LIN {X 0,Y 573.278,Z 350.069,A -85,B 0,C 180,E1 -2306.518,E2 -2306.518} C_VEL
LIN {X 0,Y 573.237,Z 350.076,A -85,B 0,C 180,E1 -2309.114,E2 -2309.114} C_VEL
LIN {X 0,Y 573.257,Z 350.077,A -85,B 0,C 180,E1 -2311.968,E2 -2311.968} C_VEL
LIN {X 0,Y 573.248,Z 350.072,A -85,B 0,C 180,E1 -2314.59,E2 -2314.59} C_VEL
LIN {X 0,Y 573.231,Z 350.084,A -85,B 0,C 180,E1 -2317.662,E2 -2317.662} C_VEL
LIN {X 0,Y 573.249,Z 350.078,A -85,B 0,C 180,E1 -2319.923,E2 -2319.923} C_VEL
LIN {X 0,Y 573.255,Z 350.073,A -85,B 0,C 180,E1 -2322.988,E2 -2322.988} C_VEL
LIN {X 0,Y 573.263,Z 350.076,A -85,B 0,C 180,E1 -2325.807,E2 -2325.807} C_VEL
LIN {X 0,Y 573.273,Z 350.07,A -85,B 0,C 180,E1 -2328.734,E2 -2328.734} C_VEL
LIN {X 0,Y 573.299,Z 350.074,A -85,B 0,C 180,E1 -2331.541,E2 -2331.541} C_VEL
LIN {X 0,Y 573.285,Z 350.068,A -85,B 0,C 180,E1 -2334.372,E2 -2334.372} C_VEL
LIN {X 0,Y 573.301,Z 350.068,A -85,B 0,C 180,E1 -2337.893,E2 -2337.893} C_VEL
LIN {X 0,Y 573.331,Z 350.064,A -85,B 0,C 180,E1 -2340.703,E2 -2340.703} C_VEL
LIN {X 0,Y 573.238,Z 350.08,A -85,B 0,C 180,E1 -2343.515,E2 -2343.515} C_VEL
LIN {X 0,Y 573.289,Z 350.072,A -85,B 0,C 180,E1 -2345.628,E2 -2345.628} C_VEL
LIN {X 0,Y 573.3,Z 350.067,A -85,B 0,C 180,E1 -2348.459,E2 -2348.459} C_VEL
LIN {X 0,Y 573.29,Z 350.075,A -85,B 0,C 180,E1 -2351.312,E2 -2351.312} C_VEL
LIN {X 0,Y 573.272,Z 350.071,A -85,B 0,C 180,E1 -2354.425,E2 -2354.425} C_VEL
LIN {X 0,Y 573.253,Z 350.082,A -85,B 0,C 180,E1 -2357.112,E2 -2357.112} C_VEL
LIN {X 0,Y 573.251,Z 350.072,A -85,B 0,C 180,E1 -2360.077,E2 -2360.077} C_VEL
LIN {X 0,Y 573.264,Z 350.078,A -85,B 0,C 180,E1 -2363.154,E2 -2363.154} C_VEL
LIN {X 0,Y 573.248,Z 350.074,A -85,B 0,C 180,E1 -2364.404,E2 -2364.404} C_VEL
LIN {X 0,Y 572.617,Z 350.161,A -85,B 0,C 180,E1 -2364.99,E2 -2364.99} C_VEL
LIN {X 0,Y 569.778,Z 350.515,A -85,B 0,C 180,E1 -2365.942,E2 -2365.942} C_VEL
LIN {X 0,Y 567.353,Z 350.815,A -85,B 0,C 180,E1 -2366.708,E2 -2366.708} C_VEL
LIN {X 0,Y 566.302,Z 350.944,A -85,B 0,C 180,E1 -2367.299,E2 -2367.299} C_VEL
LIN {X 0,Y 566.212,Z 350.952,A -85,B 0,C 180,E1 -2367.5,E2 -2367.5} C_VEL
LIN {X 0,Y 566.184,Z 350.958,A -85,B 0,C 180,E1 -2370.593,E2 -2370.593} C_VEL
LIN {X 0,Y 566.224,Z 350.953,A -85,B 0,C 180,E1 -2373.102,E2 -2373.102} C_VEL
LIN {X 0,Y 566.208,Z 350.951,A -85,B 0,C 180,E1 -2375.689,E2 -2375.689} C_VEL
LIN {X 0,Y 566.213,Z 350.955,A -85,B 0,C 180,E1 -2378.56,E2 -2378.56} C_VEL
LIN {X 0,Y 566.209,Z 350.954,A -85,B 0,C 180,E1 -2381.137,E2 -2381.137} C_VEL
LIN {X 0,Y 566.199,Z 350.953,A -85,B 0,C 180,E1 -2384.036,E2 -2384.036} C_VEL
LIN {X 0,Y 566.203,Z 350.955,A -85,B 0,C 180,E1 -2387.083,E2 -2387.083} C_VEL
LIN {X 0,Y 566.227,Z 350.949,A -85,B 0,C 180,E1 -2389.804,E2 -2389.804} C_VEL
LIN {X 0,Y 566.199,Z 350.962,A -85,B 0,C 180,E1 -2392.6,E2 -2392.6} C_VEL
LIN {X 0,Y 566.277,Z 351.069,A -85,B 0,C 180,E1 -2395.593,E2 -2395.593} C_VEL
LIN {X 0,Y 566.349,Z 357.943,A -85,B 0,C 180,E1 -2396.907,E2 -2396.907} C_VEL
LIN {X 0,Y 566.272,Z 373.418,A -85,B 0,C 180,E1 -2399.826,E2 -2399.826} C_VEL
LIN {X 0,Y 566.238,Z 374.613,A -85,B 0,C 180,E1 -2400.049,E2 -2400.049} C_VEL
LIN {X 0,Y 567.194,Z 381.693,A -85,B 0,C 180,E1 -2400.172,E2 -2400.172} C_VEL
LIN {X 0,Y 566.953,Z 481.195,A -85,B 0,C 180,E1 -2401.453,E2 -2401.453} C_VEL
LIN {X 0,Y 566.809,Z 494.766,A -85,B 0,C 180,E1 -2401.78,E2 -2401.78} C_VEL
LIN {X 0,Y 566.75,Z 507.497,A -85,B 0,C 180,E1 -2402.239,E2 -2402.239} C_VEL
LIN {X 0,Y 566.582,Z 518.434,A -85,B 0,C 180,E1 -2402.768,E2 -2402.768} C_VEL
LIN {X 0,Y 566.484,Z 529.803,A -85,B 0,C 180,E1 -2403.473,E2 -2403.473} C_VEL
LIN {X 0,Y 566.32,Z 539.973,A -85,B 0,C 180,E1 -2404.257,E2 -2404.257} C_VEL
LIN {X 0,Y 566.196,Z 548.312,A -85,B 0,C 180,E1 -2405.038,E2 -2405.038} C_VEL
LIN {X 0,Y 566.102,Z 556.91,A -85,B 0,C 180,E1 -2406.01,E2 -2406.01} C_VEL
LIN {X 0,Y 566.043,Z 564.378,A -85,B 0,C 180,E1 -2407.053,E2 -2407.053} C_VEL
LIN {X 0,Y 565.962,Z 570.591,A -85,B 0,C 180,E1 -2408.129,E2 -2408.129} C_VEL
LIN {X 0,Y 565.903,Z 575.802,A -85,B 0,C 180,E1 -2409.272,E2 -2409.272} C_VEL
LIN {X 0,Y 565.869,Z 579.731,A -85,B 0,C 180,E1 -2410.408,E2 -2410.408} C_VEL
LIN {X 0,Y 565.855,Z 581.723,A -85,B 0,C 180,E1 -2411.161,E2 -2411.161} C_VEL
LIN {X 0,Y 565.839,Z 583.2,A -85,B 0,C 180,E1 -2411.91,E2 -2411.91} C_VEL
LIN {X 0,Y 565.858,Z 584.57,A -85,B 0,C 180,E1 -2413.01,E2 -2413.01} C_VEL
LIN {X 0,Y 565.812,Z 584.985,A -85,B 0,C 180,E1 -2414.142,E2 -2414.142} C_VEL
LIN {X 0,Y 565.807,Z 584.704,A -85,B 0,C 180,E1 -2414.88,E2 -2414.88} C_VEL
LIN {X 0,Y 565.855,Z 583.986,A -85,B 0,C 180,E1 -2415.645,E2 -2415.645} C_VEL
LIN {X 0,Y 565.867,Z 582.912,A -85,B 0,C 180,E1 -2416.351,E2 -2416.351} C_VEL
LIN {X 0,Y 565.879,Z 580.421,A -85,B 0,C 180,E1 -2417.447,E2 -2417.447} C_VEL
LIN {X 0,Y 565.917,Z 576.904,A -85,B 0,C 180,E1 -2418.539,E2 -2418.539} C_VEL
LIN {X 0,Y 565.931,Z 572.283,A -85,B 0,C 180,E1 -2419.627,E2 -2419.627} C_VEL
LIN {X 0,Y 565.993,Z 565.294,A -85,B 0,C 180,E1 -2420.891,E2 -2420.891} C_VEL
LIN {X 0,Y 566.112,Z 557.744,A -85,B 0,C 180,E1 -2421.972,E2 -2421.972} C_VEL
LIN {X 0,Y 566.169,Z 550.08,A -85,B 0,C 180,E1 -2422.87,E2 -2422.87} C_VEL
LIN {X 0,Y 566.319,Z 540.76,A -85,B 0,C 180,E1 -2423.766,E2 -2423.766} C_VEL
LIN {X 0,Y 566.44,Z 530.463,A -85,B 0,C 180,E1 -2424.572,E2 -2424.572} C_VEL
LIN {X 0,Y 566.547,Z 519.075,A -85,B 0,C 180,E1 -2425.286,E2 -2425.286} C_VEL
LIN {X 0,Y 566.732,Z 507.128,A -85,B 0,C 180,E1 -2425.867,E2 -2425.867} C_VEL
LIN {X 0,Y 566.819,Z 493.96,A -85,B 0,C 180,E1 -2426.335,E2 -2426.335} C_VEL
LIN {X 0,Y 566.934,Z 480.736,A -85,B 0,C 180,E1 -2426.647,E2 -2426.647} C_VEL
LIN {X 0,Y 567.081,Z 379.638,A -85,B 0,C 180,E1 -2427.947,E2 -2427.947} C_VEL
LIN {X 0,Y 566.248,Z 374.594,A -85,B 0,C 180,E1 -2428.044,E2 -2428.044} C_VEL
LIN {X 0,Y 566.341,Z 358.556,A -85,B 0,C 180,E1 -2431.067,E2 -2431.067} C_VEL
LIN {X 0,Y 566.465,Z 352.939,A -85,B 0,C 180,E1 -2432.133,E2 -2432.133} C_VEL
LIN {X 0,Y 566.263,Z 350.949,A -85,B 0,C 180,E1 -2432.534,E2 -2432.534} C_VEL
LIN {X 0,Y 566.262,Z 350.95,A -85,B 0,C 180,E1 -2435.698,E2 -2435.698} C_VEL
LIN {X 0,Y 566.212,Z 350.95,A -85,B 0,C 180,E1 -2438.566,E2 -2438.566} C_VEL
LIN {X 0,Y 566.249,Z 350.954,A -85,B 0,C 180,E1 -2441.454,E2 -2441.454} C_VEL
LIN {X 0,Y 566.241,Z 350.946,A -85,B 0,C 180,E1 -2444.506,E2 -2444.506} C_VEL
LIN {X 0,Y 566.205,Z 350.961,A -85,B 0,C 180,E1 -2447.331,E2 -2447.331} C_VEL
LIN {X 0,Y 566.212,Z 350.949,A -85,B 0,C 180,E1 -2450.337,E2 -2450.337} C_VEL
LIN {X 0,Y 566.194,Z 350.959,A -85,B 0,C 180,E1 -2453.403,E2 -2453.403} C_VEL
LIN {X 0,Y 566.218,Z 350.951,A -85,B 0,C 180,E1 -2455.748,E2 -2455.748} C_VEL
LIN {X 0,Y 566.205,Z 350.95,A -85,B 0,C 180,E1 -2458.201,E2 -2458.201} C_VEL
LIN {X 0,Y 566.202,Z 350.959,A -85,B 0,C 180,E1 -2461.077,E2 -2461.077} C_VEL
LIN {X 0,Y 566.214,Z 350.951,A -85,B 0,C 180,E1 -2463.733,E2 -2463.733} C_VEL
LIN {X 0,Y 566.218,Z 350.951,A -85,B 0,C 180,E1 -2466.568,E2 -2466.568} C_VEL
LIN {X 0,Y 566.213,Z 350.951,A -85,B 0,C 180,E1 -2469.685,E2 -2469.685} C_VEL
LIN {X 0,Y 566.213,Z 350.949,A -85,B 0,C 180,E1 -2472.086,E2 -2472.086} C_VEL
LIN {X 0,Y 566.172,Z 350.965,A -85,B 0,C 180,E1 -2475.035,E2 -2475.035} C_VEL
LIN {X 0,Y 566.214,Z 350.949,A -85,B 0,C 180,E1 -2477.912,E2 -2477.912} C_VEL
LIN {X 0,Y 566.219,Z 350.955,A -85,B 0,C 180,E1 -2480.726,E2 -2480.726} C_VEL
LIN {X 0,Y 566.214,Z 350.949,A -85,B 0,C 180,E1 -2483.782,E2 -2483.782} C_VEL
LIN {X 0,Y 566.207,Z 350.951,A -85,B 0,C 180,E1 -2486.265,E2 -2486.265} C_VEL
LIN {X 0,Y 566.195,Z 350.961,A -85,B 0,C 180,E1 -2488.921,E2 -2488.921} C_VEL
LIN {X 0,Y 566.222,Z 350.948,A -85,B 0,C 180,E1 -2491.858,E2 -2491.858} C_VEL
LIN {X 0,Y 566.219,Z 350.951,A -85,B 0,C 180,E1 -2494.251,E2 -2494.251} C_VEL
LIN {X 0,Y 566.186,Z 350.962,A -85,B 0,C 180,E1 -2496.712,E2 -2496.712} C_VEL
LIN {X 0,Y 566.213,Z 350.949,A -85,B 0,C 180,E1 -2499.662,E2 -2499.662} C_VEL
LIN {X 0,Y 566.198,Z 350.961,A -85,B 0,C 180,E1 -2502.668,E2 -2502.668} C_VEL
LIN {X 0,Y 566.225,Z 350.948,A -85,B 0,C 180,E1 -2505.626,E2 -2505.626} C_VEL
LIN {X 0,Y 566.266,Z 350.953,A -85,B 0,C 180,E1 -2508.654,E2 -2508.654} C_VEL
LIN {X 0,Y 566.24,Z 350.946,A -85,B 0,C 180,E1 -2511.434,E2 -2511.434} C_VEL
LIN {X 0,Y 566.253,Z 350.95,A -85,B 0,C 180,E1 -2514.301,E2 -2514.301} C_VEL
LIN {X 0,Y 566.272,Z 350.943,A -85,B 0,C 180,E1 -2517.866,E2 -2517.866} C_VEL
LIN {X 0,Y 566.299,Z 350.945,A -85,B 0,C 180,E1 -2520.711,E2 -2520.711} C_VEL
LIN {X 0,Y 566.27,Z 350.946,A -85,B 0,C 180,E1 -2522.845,E2 -2522.845} C_VEL
LIN {X 0,Y 566.252,Z 350.945,A -85,B 0,C 180,E1 -2525.698,E2 -2525.698} C_VEL
LIN {X 0,Y 566.239,Z 350.954,A -85,B 0,C 180,E1 -2528.565,E2 -2528.565} C_VEL
LIN {X 0,Y 566.241,Z 350.946,A -85,B 0,C 180,E1 -2531.454,E2 -2531.454} C_VEL
LIN {X 0,Y 566.224,Z 350.956,A -85,B 0,C 180,E1 -2534.507,E2 -2534.507} C_VEL
LIN {X 0,Y 566.196,Z 350.951,A -85,B 0,C 180,E1 -2537.332,E2 -2537.332} C_VEL
LIN {X 0,Y 566.212,Z 350.959,A -85,B 0,C 180,E1 -2540.337,E2 -2540.337} C_VEL
LIN {X 0,Y 566.182,Z 350.953,A -85,B 0,C 180,E1 -2543.404,E2 -2543.404} C_VEL
LIN {X 0,Y 566.217,Z 350.951,A -85,B 0,C 180,E1 -2545.749,E2 -2545.749} C_VEL
LIN {X 0,Y 566.2,Z 350.961,A -85,B 0,C 180,E1 -2548.204,E2 -2548.204} C_VEL
LIN {X 0,Y 566.187,Z 350.956,A -85,B 0,C 180,E1 -2550.592,E2 -2550.592} C_VEL
LIN {X 0,Y 566.222,Z 350.948,A -85,B 0,C 180,E1 -2553.102,E2 -2553.102} C_VEL
LIN {X 0,Y 566.205,Z 350.953,A -85,B 0,C 180,E1 -2555.689,E2 -2555.689} C_VEL
LIN {X 0,Y 566.211,Z 350.952,A -85,B 0,C 180,E1 -2558.56,E2 -2558.56} C_VEL
LIN {X 0,Y 566.208,Z 350.95,A -85,B 0,C 180,E1 -2561.137,E2 -2561.137} C_VEL
LIN {X 0,Y 566.196,Z 350.962,A -85,B 0,C 180,E1 -2564.036,E2 -2564.036} C_VEL
LIN {X 0,Y 566.201,Z 350.951,A -85,B 0,C 180,E1 -2567.083,E2 -2567.083} C_VEL
LIN {X 0,Y 566.225,Z 350.955,A -85,B 0,C 180,E1 -2569.804,E2 -2569.804} C_VEL
LIN {X 0,Y 566.197,Z 350.952,A -85,B 0,C 180,E1 -2572.6,E2 -2572.6} C_VEL
LIN {X 0,Y 566.221,Z 350.949,A -85,B 0,C 180,E1 -2575.184,E2 -2575.184} C_VEL
LIN {X 0,Y 566.234,Z 350.954,A -85,B 0,C 180,E1 -2577.744,E2 -2577.744} C_VEL
LIN {X 0,Y 566.228,Z 350.952,A -85,B 0,C 180,E1 -2580.324,E2 -2580.324} C_VEL
LIN {X 0,Y 566.219,Z 350.951,A -85,B 0,C 180,E1 -2582.662,E2 -2582.662} C_VEL
LIN {X 0,Y 566.237,Z 350.95,A -85,B 0,C 180,E1 -2585.04,E2 -2585.04} C_VEL
LIN {X 0,Y 566.233,Z 351.027,A -85,B 0,C 180,E1 -2585.919,E2 -2585.919} C_VEL
LIN {X 0,Y 567.201,Z 357.146,A -85,B 0,C 180,E1 -2586.834,E2 -2586.834} C_VEL
LIN {X 0,Y 566.963,Z 376.072,A -85,B 0,C 180,E1 -2589.502,E2 -2589.502} C_VEL
LIN {X 0,Y 566.667,Z 397.345,A -85,B 0,C 180,E1 -2592.497,E2 -2592.497} C_VEL
LIN {X 0,Y 566.459,Z 419.948,A -85,B 0,C 180,E1 -2595.633,E2 -2595.633} C_VEL
LIN {X 0,Y 566.417,Z 422.524,A -85,B 0,C 180,E1 -2595.987,E2 -2595.987} C_VEL
LIN {X 0,Y 567.226,Z 430.323,A -85,B 0,C 180,E1 -2596.11,E2 -2596.11} C_VEL
LIN {X 0,Y 566.964,Z 530.961,A -85,B 0,C 180,E1 -2597.403,E2 -2597.403} C_VEL
LIN {X 0,Y 566.871,Z 544.228,A -85,B 0,C 180,E1 -2597.72,E2 -2597.72} C_VEL
LIN {X 0,Y 566.74,Z 556.383,A -85,B 0,C 180,E1 -2598.148,E2 -2598.148} C_VEL
LIN {X 0,Y 566.589,Z 568.449,A -85,B 0,C 180,E1 -2598.724,E2 -2598.724} C_VEL
LIN {X 0,Y 566.442,Z 580.203,A -85,B 0,C 180,E1 -2599.455,E2 -2599.455} C_VEL
LIN {X 0,Y 566.321,Z 590.605,A -85,B 0,C 180,E1 -2600.266,E2 -2600.266} C_VEL
LIN {X 0,Y 566.207,Z 599.115,A -85,B 0,C 180,E1 -2601.074,E2 -2601.074} C_VEL
LIN {X 0,Y 566.112,Z 606.962,A -85,B 0,C 180,E1 -2601.972,E2 -2601.972} C_VEL
LIN {X 0,Y 566.003,Z 614.623,A -85,B 0,C 180,E1 -2603.047,E2 -2603.047} C_VEL
LIN {X 0,Y 566.004,Z 621.68,A -85,B 0,C 180,E1 -2604.299,E2 -2604.299} C_VEL
LIN {X 0,Y 565.933,Z 626.373,A -85,B 0,C 180,E1 -2605.37,E2 -2605.37} C_VEL
LIN {X 0,Y 565.927,Z 629.958,A -85,B 0,C 180,E1 -2606.44,E2 -2606.44} C_VEL
LIN {X 0,Y 565.878,Z 631.808,A -85,B 0,C 180,E1 -2607.153,E2 -2607.153} C_VEL
LIN {X 0,Y 565.846,Z 634.185,A -85,B 0,C 180,E1 -2608.577,E2 -2608.577} C_VEL
LIN {X 0,Y 565.839,Z 635,A -85,B 0,C 180,E1 -2610,E2 -2610} C_VEL
LIN {X 0,Y 565.846,Z 634.186,A -85,B 0,C 180,E1 -2611.423,E2 -2611.423} C_VEL
LIN {X 0,Y 565.878,Z 631.81,A -85,B 0,C 180,E1 -2612.847,E2 -2612.847} C_VEL
LIN {X 0,Y 565.926,Z 628.896,A -85,B 0,C 180,E1 -2613.916,E2 -2613.916} C_VEL
LIN {X 0,Y 565.878,Z 624.949,A -85,B 0,C 180,E1 -2614.987,E2 -2614.987} C_VEL
LIN {X 0,Y 566.002,Z 619.868,A -85,B 0,C 180,E1 -2616.058,E2 -2616.058} C_VEL
LIN {X 0,Y 566.04,Z 613.469,A -85,B 0,C 180,E1 -2617.132,E2 -2617.132} C_VEL
LIN {X 0,Y 566.133,Z 605.479,A -85,B 0,C 180,E1 -2618.207,E2 -2618.207} C_VEL
LIN {X 0,Y 566.228,Z 597.337,A -85,B 0,C 180,E1 -2619.105,E2 -2619.105} C_VEL
LIN {X 0,Y 566.343,Z 587.403,A -85,B 0,C 180,E1 -2620.005,E2 -2620.005} C_VEL
LIN {X 0,Y 566.529,Z 576.294,A -85,B 0,C 180,E1 -2620.807,E2 -2620.807} C_VEL
LIN {X 0,Y 566.612,Z 565.181,A -85,B 0,C 180,E1 -2621.446,E2 -2621.446} C_VEL
LIN {X 0,Y 566.736,Z 552.989,A -85,B 0,C 180,E1 -2621.988,E2 -2621.988} C_VEL
LIN {X 0,Y 566.91,Z 540.187,A -85,B 0,C 180,E1 -2622.393,E2 -2622.393} C_VEL
LIN {X 0,Y 566.997,Z 528.125,A -85,B 0,C 180,E1 -2622.641,E2 -2622.641} C_VEL
LIN {X 0,Y 567.065,Z 426.951,A -85,B 0,C 180,E1 -2623.937,E2 -2623.937} C_VEL
LIN {X 0,Y 566.435,Z 422.441,A -85,B 0,C 180,E1 -2624.024,E2 -2624.024} C_VEL
LIN {X 0,Y 566.648,Z 399.148,A -85,B 0,C 180,E1 -2627.251,E2 -2627.251} C_VEL
LIN {X 0,Y 566.926,Z 378.732,A -85,B 0,C 180,E1 -2630.121,E2 -2630.121} C_VEL
LIN {X 0,Y 567.199,Z 357.118,A -85,B 0,C 180,E1 -2633.166,E2 -2633.166} C_VEL
LIN {X 0,Y 566.236,Z 350.957,A -85,B 0,C 180,E1 -2634.105,E2 -2634.105} C_VEL
LIN {X 0,Y 566.209,Z 350.954,A -85,B 0,C 180,E1 -2636.659,E2 -2636.659} C_VEL
LIN {X 0,Y 566.196,Z 350.953,A -85,B 0,C 180,E1 -2638.952,E2 -2638.952} C_VEL
LIN {X 0,Y 566.203,Z 350.952,A -85,B 0,C 180,E1 -2641.42,E2 -2641.42} C_VEL
LIN {X 0,Y 566.212,Z 350.957,A -85,B 0,C 180,E1 -2643.955,E2 -2643.955} C_VEL
LIN {X 0,Y 566.215,Z 350.952,A -85,B 0,C 180,E1 -2646.568,E2 -2646.568} C_VEL
LIN {X 0,Y 566.212,Z 350.954,A -85,B 0,C 180,E1 -2649.685,E2 -2649.685} C_VEL
LIN {X 0,Y 566.211,Z 350.957,A -85,B 0,C 180,E1 -2652.086,E2 -2652.086} C_VEL
LIN {X 0,Y 566.169,Z 350.955,A -85,B 0,C 180,E1 -2655.035,E2 -2655.035} C_VEL
LIN {X 0,Y 566.214,Z 350.956,A -85,B 0,C 180,E1 -2658.135,E2 -2658.135} C_VEL
LIN {X 0,Y 566.218,Z 350.949,A -85,B 0,C 180,E1 -2660.727,E2 -2660.727} C_VEL
LIN {X 0,Y 566.211,Z 350.959,A -85,B 0,C 180,E1 -2663.783,E2 -2663.783} C_VEL
LIN {X 0,Y 566.222,Z 350.95,A -85,B 0,C 180,E1 -2666.262,E2 -2666.262} C_VEL
LIN {X 0,Y 566.196,Z 350.952,A -85,B 0,C 180,E1 -2668.921,E2 -2668.921} C_VEL
LIN {X 0,Y 566.189,Z 350.953,A -85,B 0,C 180,E1 -2671.046,E2 -2671.046} C_VEL
LIN {X 0,Y 566.237,Z 350.953,A -85,B 0,C 180,E1 -2673.46,E2 -2673.46} C_VEL
LIN {X 0,Y 566.19,Z 350.96,A -85,B 0,C 180,E1 -2675.819,E2 -2675.819} C_VEL
LIN {X 0,Y 566.208,Z 350.95,A -85,B 0,C 180,E1 -2678.902,E2 -2678.902} C_VEL
LIN {X 0,Y 566.205,Z 350.954,A -85,B 0,C 180,E1 -2681.172,E2 -2681.172} C_VEL
LIN {X 0,Y 566.213,Z 350.956,A -85,B 0,C 180,E1 -2683.412,E2 -2683.412} C_VEL
LIN {X 0,Y 566.191,Z 350.952,A -85,B 0,C 180,E1 -2686.359,E2 -2686.359} C_VEL
LIN {X 0,Y 566.265,Z 350.943,A -85,B 0,C 180,E1 -2688.654,E2 -2688.654} C_VEL
LIN {X 0,Y 566.241,Z 350.955,A -85,B 0,C 180,E1 -2691.435,E2 -2691.435} C_VEL
LIN {X 0,Y 566.253,Z 350.945,A -85,B 0,C 180,E1 -2694.302,E2 -2694.302} C_VEL
LIN {X 0,Y 566.272,Z 350.944,A -85,B 0,C 180,E1 -2697.866,E2 -2697.866} C_VEL
LIN {X 0,Y 566.3,Z 350.94,A -85,B 0,C 180,E1 -2700.711,E2 -2700.711} C_VEL
LIN {X 0,Y 566.272,Z 350.944,A -85,B 0,C 180,E1 -2702.846,E2 -2702.846} C_VEL
LIN {X 0,Y 566.256,Z 350.947,A -85,B 0,C 180,E1 -2705.699,E2 -2705.699} C_VEL
LIN {X 0,Y 566.242,Z 350.946,A -85,B 0,C 180,E1 -2708.566,E2 -2708.566} C_VEL
LIN {X 0,Y 566.242,Z 350.95,A -85,B 0,C 180,E1 -2711.455,E2 -2711.455} C_VEL
LIN {X 0,Y 566.225,Z 350.949,A -85,B 0,C 180,E1 -2714.508,E2 -2714.508} C_VEL
LIN {X 0,Y 566.197,Z 350.958,A -85,B 0,C 180,E1 -2717.332,E2 -2717.332} C_VEL
LIN {X 0,Y 566.213,Z 350.949,A -85,B 0,C 180,E1 -2720.337,E2 -2720.337} C_VEL
LIN {X 0,Y 566.223,Z 350.951,A -85,B 0,C 180,E1 -2723.403,E2 -2723.403} C_VEL
LIN {X 0,Y 566.219,Z 350.949,A -85,B 0,C 180,E1 -2725.749,E2 -2725.749} C_VEL
LIN {X 0,Y 566.212,Z 350.952,A -85,B 0,C 180,E1 -2727.5,E2 -2727.5} C_VEL
LIN {X 0,Y 565.531,Z 351.036,A -85,B 0,C 180,E1 -2728.093,E2 -2728.093} C_VEL
LIN {X 0,Y 562.66,Z 351.4,A -85,B 0,C 180,E1 -2729.057,E2 -2729.057} C_VEL
LIN {X 0,Y 560.246,Z 351.696,A -85,B 0,C 180,E1 -2729.832,E2 -2729.832} C_VEL
LIN {X 0,Y 559.22,Z 351.823,A -85,B 0,C 180,E1 -2730.431,E2 -2730.431} C_VEL
LIN {X 0,Y 559.141,Z 351.834,A -85,B 0,C 180,E1 -2730.633,E2 -2730.633} C_VEL
LIN {X 0,Y 559.173,Z 351.826,A -85,B 0,C 180,E1 -2733.575,E2 -2733.575} C_VEL
LIN {X 0,Y 559.165,Z 351.831,A -85,B 0,C 180,E1 -2736.45,E2 -2736.45} C_VEL
LIN {X 0,Y 559.175,Z 351.834,A -85,B 0,C 180,E1 -2738.935,E2 -2738.935} C_VEL
LIN {X 0,Y 559.19,Z 351.824,A -85,B 0,C 180,E1 -2741.768,E2 -2741.768} C_VEL
LIN {X 0,Y 559.138,Z 351.839,A -85,B 0,C 180,E1 -2744.74,E2 -2744.74} C_VEL
LIN {X 0,Y 559.162,Z 351.83,A -85,B 0,C 180,E1 -2747.258,E2 -2747.258} C_VEL
LIN {X 0,Y 559.185,Z 351.828,A -85,B 0,C 180,E1 -2750.136,E2 -2750.136} C_VEL
LIN {X 0,Y 559.148,Z 351.838,A -85,B 0,C 180,E1 -2752.893,E2 -2752.893} C_VEL
LIN {X 0,Y 559.244,Z 351.992,A -85,B 0,C 180,E1 -2755.508,E2 -2755.508} C_VEL
LIN {X 0,Y 559.399,Z 356.695,A -85,B 0,C 180,E1 -2756.442,E2 -2756.442} C_VEL
LIN {X 0,Y 559.231,Z 372.166,A -85,B 0,C 180,E1 -2759.405,E2 -2759.405} C_VEL
LIN {X 0,Y 559.235,Z 374.729,A -85,B 0,C 180,E1 -2759.88,E2 -2759.88} C_VEL
LIN {X 0,Y 560.319,Z 382.315,A -85,B 0,C 180,E1 -2760.006,E2 -2760.006} C_VEL
LIN {X 0,Y 560.027,Z 481.111,A -85,B 0,C 180,E1 -2761.293,E2 -2761.293} C_VEL
LIN {X 0,Y 559.88,Z 494.363,A -85,B 0,C 180,E1 -2761.613,E2 -2761.613} C_VEL
LIN {X 0,Y 559.789,Z 506.94,A -85,B 0,C 180,E1 -2762.067,E2 -2762.067} C_VEL
LIN {X 0,Y 559.605,Z 518.268,A -85,B 0,C 180,E1 -2762.616,E2 -2762.616} C_VEL
LIN {X 0,Y 559.477,Z 529.474,A -85,B 0,C 180,E1 -2763.316,E2 -2763.316} C_VEL
LIN {X 0,Y 559.31,Z 539.707,A -85,B 0,C 180,E1 -2764.11,E2 -2764.11} C_VEL
LIN {X 0,Y 559.157,Z 548.987,A -85,B 0,C 180,E1 -2764.993,E2 -2764.993} C_VEL
LIN {X 0,Y 559.052,Z 556.727,A -85,B 0,C 180,E1 -2765.886,E2 -2765.886} C_VEL
LIN {X 0,Y 558.971,Z 563.554,A -85,B 0,C 180,E1 -2766.835,E2 -2766.835} C_VEL
LIN {X 0,Y 558.902,Z 569.486,A -85,B 0,C 180,E1 -2767.838,E2 -2767.838} C_VEL
LIN {X 0,Y 558.843,Z 574.96,A -85,B 0,C 180,E1 -2768.998,E2 -2768.998} C_VEL
LIN {X 0,Y 558.816,Z 579.106,A -85,B 0,C 180,E1 -2770.15,E2 -2770.15} C_VEL
LIN {X 0,Y 558.782,Z 581.205,A -85,B 0,C 180,E1 -2770.913,E2 -2770.913} C_VEL
LIN {X 0,Y 558.735,Z 582.842,A -85,B 0,C 180,E1 -2771.672,E2 -2771.672} C_VEL
LIN {X 0,Y 558.767,Z 584.519,A -85,B 0,C 180,E1 -2772.923,E2 -2772.923} C_VEL
LIN {X 0,Y 558.729,Z 584.982,A -85,B 0,C 180,E1 -2773.935,E2 -2773.935} C_VEL
LIN {X 0,Y 558.71,Z 584.839,A -85,B 0,C 180,E1 -2774.683,E2 -2774.683} C_VEL
LIN {X 0,Y 558.762,Z 584.079,A -85,B 0,C 180,E1 -2775.581,E2 -2775.581} C_VEL
LIN {X 0,Y 558.751,Z 581.839,A -85,B 0,C 180,E1 -2776.915,E2 -2776.915} C_VEL
LIN {X 0,Y 558.824,Z 578.857,A -85,B 0,C 180,E1 -2778.024,E2 -2778.024} C_VEL
LIN {X 0,Y 558.853,Z 574.823,A -85,B 0,C 180,E1 -2779.127,E2 -2779.127} C_VEL
LIN {X 0,Y 558.889,Z 568.615,A -85,B 0,C 180,E1 -2780.409,E2 -2780.409} C_VEL
LIN {X 0,Y 558.983,Z 561.861,A -85,B 0,C 180,E1 -2781.505,E2 -2781.505} C_VEL
LIN {X 0,Y 559.077,Z 553.51,A -85,B 0,C 180,E1 -2782.597,E2 -2782.597} C_VEL
LIN {X 0,Y 559.218,Z 544.931,A -85,B 0,C 180,E1 -2783.506,E2 -2783.506} C_VEL
LIN {X 0,Y 559.391,Z 534.401,A -85,B 0,C 180,E1 -2784.412,E2 -2784.412} C_VEL
LIN {X 0,Y 559.502,Z 524.009,A -85,B 0,C 180,E1 -2785.136,E2 -2785.136} C_VEL
LIN {X 0,Y 559.737,Z 512.524,A -85,B 0,C 180,E1 -2785.77,E2 -2785.77} C_VEL
LIN {X 0,Y 559.814,Z 500.752,A -85,B 0,C 180,E1 -2786.266,E2 -2786.266} C_VEL
LIN {X 0,Y 559.938,Z 488.019,A -85,B 0,C 180,E1 -2786.65,E2 -2786.65} C_VEL
LIN {X 0,Y 560.062,Z 474.623,A -85,B 0,C 180,E1 -2786.898,E2 -2786.898} C_VEL
LIN {X 0,Y 560.162,Z 380.375,A -85,B 0,C 180,E1 -2788.113,E2 -2788.113} C_VEL
LIN {X 0,Y 559.222,Z 374.602,A -85,B 0,C 180,E1 -2788.222,E2 -2788.222} C_VEL
LIN {X 0,Y 559.318,Z 359.631,A -85,B 0,C 180,E1 -2791.08,E2 -2791.08} C_VEL
LIN {X 0,Y 559.294,Z 352.312,A -85,B 0,C 180,E1 -2792.521,E2 -2792.521} C_VEL
LIN {X 0,Y 559.244,Z 351.825,A -85,B 0,C 180,E1 -2792.656,E2 -2792.656} C_VEL
LIN {X 0,Y 559.23,Z 351.825,A -85,B 0,C 180,E1 -2795.77,E2 -2795.77} C_VEL
LIN {X 0,Y 559.177,Z 351.827,A -85,B 0,C 180,E1 -2798.674,E2 -2798.674} C_VEL
LIN {X 0,Y 559.212,Z 351.828,A -85,B 0,C 180,E1 -2801.6,E2 -2801.6} C_VEL
LIN {X 0,Y 559.206,Z 351.823,A -85,B 0,C 180,E1 -2804.595,E2 -2804.595} C_VEL
LIN {X 0,Y 559.164,Z 351.834,A -85,B 0,C 180,E1 -2807.556,E2 -2807.556} C_VEL
LIN {X 0,Y 559.171,Z 351.829,A -85,B 0,C 180,E1 -2809.837,E2 -2809.837} C_VEL
LIN {X 0,Y 559.145,Z 351.83,A -85,B 0,C 180,E1 -2812.152,E2 -2812.152} C_VEL
LIN {X 0,Y 559.183,Z 351.834,A -85,B 0,C 180,E1 -2815.186,E2 -2815.186} C_VEL
LIN {X 0,Y 559.16,Z 351.831,A -85,B 0,C 180,E1 -2817.713,E2 -2817.713} C_VEL
LIN {X 0,Y 559.159,Z 351.828,A -85,B 0,C 180,E1 -2820.182,E2 -2820.182} C_VEL
LIN {X 0,Y 559.177,Z 351.829,A -85,B 0,C 180,E1 -2822.713,E2 -2822.713} C_VEL
LIN {X 0,Y 559.16,Z 351.835,A -85,B 0,C 180,E1 -2825.321,E2 -2825.321} C_VEL
LIN {X 0,Y 559.136,Z 351.831,A -85,B 0,C 180,E1 -2828.016,E2 -2828.016} C_VEL
LIN {X 0,Y 559.176,Z 351.831,A -85,B 0,C 180,E1 -2830.81,E2 -2830.81} C_VEL
LIN {X 0,Y 559.143,Z 351.831,A -85,B 0,C 180,E1 -2833.732,E2 -2833.732} C_VEL
LIN {X 0,Y 559.169,Z 351.833,A -85,B 0,C 180,E1 -2836.8,E2 -2836.8} C_VEL
LIN {X 0,Y 559.173,Z 351.833,A -85,B 0,C 180,E1 -2839.189,E2 -2839.189} C_VEL
LIN {X 0,Y 559.132,Z 351.831,A -85,B 0,C 180,E1 -2841.982,E2 -2841.982} C_VEL
LIN {X 0,Y 559.154,Z 351.836,A -85,B 0,C 180,E1 -2844.782,E2 -2844.782} C_VEL
LIN {X 0,Y 559.17,Z 351.829,A -85,B 0,C 180,E1 -2847.36,E2 -2847.36} C_VEL
LIN {X 0,Y 559.144,Z 351.831,A -85,B 0,C 180,E1 -2850.141,E2 -2850.141} C_VEL
LIN {X 0,Y 559.177,Z 351.83,A -85,B 0,C 180,E1 -2853.169,E2 -2853.169} C_VEL
LIN {X 0,Y 559.15,Z 351.83,A -85,B 0,C 180,E1 -2855.494,E2 -2855.494} C_VEL
LIN {X 0,Y 559.17,Z 351.834,A -85,B 0,C 180,E1 -2858.623,E2 -2858.623} C_VEL
LIN {X 0,Y 559.164,Z 351.834,A -85,B 0,C 180,E1 -2860.926,E2 -2860.926} C_VEL
LIN {X 0,Y 559.165,Z 351.828,A -85,B 0,C 180,E1 -2863.948,E2 -2863.948} C_VEL
LIN {X 0,Y 559.167,Z 351.83,A -85,B 0,C 180,E1 -2866.184,E2 -2866.184} C_VEL
LIN {X 0,Y 559.202,Z 351.825,A -85,B 0,C 180,E1 -2869.133,E2 -2869.133} C_VEL
LIN {X 0,Y 559.201,Z 351.825,A -85,B 0,C 180,E1 -2872.053,E2 -2872.053} C_VEL
LIN {X 0,Y 559.251,Z 351.821,A -85,B 0,C 180,E1 -2874.953,E2 -2874.953} C_VEL
LIN {X 0,Y 559.243,Z 351.818,A -85,B 0,C 180,E1 -2877.839,E2 -2877.839} C_VEL
LIN {X 0,Y 559.268,Z 351.821,A -85,B 0,C 180,E1 -2880.72,E2 -2880.72} C_VEL
LIN {X 0,Y 559.236,Z 351.822,A -85,B 0,C 180,E1 -2882.881,E2 -2882.881} C_VEL
LIN {X 0,Y 559.221,Z 351.821,A -85,B 0,C 180,E1 -2885.77,E2 -2885.77} C_VEL
LIN {X 0,Y 559.194,Z 351.829,A -85,B 0,C 180,E1 -2888.674,E2 -2888.674} C_VEL
LIN {X 0,Y 559.199,Z 351.823,A -85,B 0,C 180,E1 -2891.6,E2 -2891.6} C_VEL
LIN {X 0,Y 559.189,Z 351.83,A -85,B 0,C 180,E1 -2894.596,E2 -2894.596} C_VEL
LIN {X 0,Y 559.155,Z 351.829,A -85,B 0,C 180,E1 -2897.557,E2 -2897.557} C_VEL
LIN {X 0,Y 559.166,Z 351.83,A -85,B 0,C 180,E1 -2899.838,E2 -2899.838} C_VEL
LIN {X 0,Y 559.136,Z 351.839,A -85,B 0,C 180,E1 -2902.153,E2 -2902.153} C_VEL
LIN {X 0,Y 559.171,Z 351.827,A -85,B 0,C 180,E1 -2905.188,E2 -2905.188} C_VEL
LIN {X 0,Y 559.187,Z 351.827,A -85,B 0,C 180,E1 -2907.712,E2 -2907.712} C_VEL
LIN {X 0,Y 559.161,Z 351.838,A -85,B 0,C 180,E1 -2910.182,E2 -2910.182} C_VEL
LIN {X 0,Y 559.169,Z 351.829,A -85,B 0,C 180,E1 -2912.714,E2 -2912.714} C_VEL
LIN {X 0,Y 559.151,Z 351.829,A -85,B 0,C 180,E1 -2915.322,E2 -2915.322} C_VEL
LIN {X 0,Y 559.13,Z 351.84,A -85,B 0,C 180,E1 -2918.018,E2 -2918.018} C_VEL
LIN {X 0,Y 559.172,Z 351.827,A -85,B 0,C 180,E1 -2920.811,E2 -2920.811} C_VEL
LIN {X 0,Y 559.158,Z 351.833,A -85,B 0,C 180,E1 -2923.732,E2 -2923.732} C_VEL
LIN {X 0,Y 559.146,Z 351.83,A -85,B 0,C 180,E1 -2926.804,E2 -2926.804} C_VEL
LIN {X 0,Y 559.174,Z 351.827,A -85,B 0,C 180,E1 -2929.19,E2 -2929.19} C_VEL
LIN {X 0,Y 559.133,Z 351.841,A -85,B 0,C 180,E1 -2931.983,E2 -2931.983} C_VEL
LIN {X 0,Y 559.159,Z 351.828,A -85,B 0,C 180,E1 -2934.784,E2 -2934.784} C_VEL
LIN {X 0,Y 559.173,Z 351.828,A -85,B 0,C 180,E1 -2937.362,E2 -2937.362} C_VEL
LIN {X 0,Y 559.189,Z 351.831,A -85,B 0,C 180,E1 -2940.136,E2 -2940.136} C_VEL
LIN {X 0,Y 559.172,Z 351.83,A -85,B 0,C 180,E1 -2943.173,E2 -2943.173} C_VEL
LIN {X 0,Y 559.198,Z 351.961,A -85,B 0,C 180,E1 -2945.769,E2 -2945.769} C_VEL
LIN {X 0,Y 560.28,Z 358.226,A -85,B 0,C 180,E1 -2946.727,E2 -2946.727} C_VEL
LIN {X 0,Y 559.998,Z 377.197,A -85,B 0,C 180,E1 -2949.427,E2 -2949.427} C_VEL
LIN {X 0,Y 559.713,Z 397.345,A -85,B 0,C 180,E1 -2952.273,E2 -2952.273} C_VEL
LIN {X 0,Y 559.463,Z 418.899,A -85,B 0,C 180,E1 -2955.303,E2 -2955.303} C_VEL
LIN {X 0,Y 559.419,Z 422.524,A -85,B 0,C 180,E1 -2955.808,E2 -2955.808} C_VEL
LIN {X 0,Y 560.336,Z 430.323,A -85,B 0,C 180,E1 -2955.936,E2 -2955.936} C_VEL
LIN {X 0,Y 560.058,Z 530.961,A -85,B 0,C 180,E1 -2957.246,E2 -2957.246} C_VEL
LIN {X 0,Y 559.927,Z 544.227,A -85,B 0,C 180,E1 -2957.565,E2 -2957.565} C_VEL
LIN {X 0,Y 559.786,Z 556.384,A -85,B 0,C 180,E1 -2957.999,E2 -2957.999} C_VEL
LIN {X 0,Y 559.615,Z 568.322,A -85,B 0,C 180,E1 -2958.574,E2 -2958.574} C_VEL
LIN {X 0,Y 559.461,Z 580.201,A -85,B 0,C 180,E1 -2959.322,E2 -2959.322} C_VEL
LIN {X 0,Y 559.301,Z 590.606,A -85,B 0,C 180,E1 -2960.142,E2 -2960.142} C_VEL
LIN {X 0,Y 559.161,Z 599.115,A -85,B 0,C 180,E1 -2960.961,E2 -2960.961} C_VEL
LIN {X 0,Y 559.05,Z 606.962,A -85,B 0,C 180,E1 -2961.87,E2 -2961.87} C_VEL
LIN {X 0,Y 558.943,Z 614.623,A -85,B 0,C 180,E1 -2962.959,E2 -2962.959} C_VEL
LIN {X 0,Y 558.935,Z 621.68,A -85,B 0,C 180,E1 -2964.227,E2 -2964.227} C_VEL
LIN {X 0,Y 558.827,Z 626.373,A -85,B 0,C 180,E1 -2965.311,E2 -2965.311} C_VEL
LIN {X 0,Y 558.836,Z 629.958,A -85,B 0,C 180,E1 -2966.395,E2 -2966.395} C_VEL
LIN {X 0,Y 558.799,Z 631.808,A -85,B 0,C 180,E1 -2967.116,E2 -2967.116} C_VEL
LIN {X 0,Y 558.745,Z 634.184,A -85,B 0,C 180,E1 -2968.559,E2 -2968.559} C_VEL
LIN {X 0,Y 558.74,Z 635,A -85,B 0,C 180,E1 -2970,E2 -2970} C_VEL
LIN {X 0,Y 558.745,Z 634.185,A -85,B 0,C 180,E1 -2971.441,E2 -2971.441} C_VEL
LIN {X 0,Y 558.799,Z 631.81,A -85,B 0,C 180,E1 -2972.884,E2 -2972.884} C_VEL
LIN {X 0,Y 558.843,Z 628.896,A -85,B 0,C 180,E1 -2973.966,E2 -2973.966} C_VEL
LIN {X 0,Y 558.799,Z 624.949,A -85,B 0,C 180,E1 -2975.051,E2 -2975.051} C_VEL
LIN {X 0,Y 558.921,Z 619.868,A -85,B 0,C 180,E1 -2976.135,E2 -2976.135} C_VEL
LIN {X 0,Y 558.977,Z 613.469,A -85,B 0,C 180,E1 -2977.223,E2 -2977.223} C_VEL
LIN {X 0,Y 559.098,Z 605.479,A -85,B 0,C 180,E1 -2978.311,E2 -2978.311} C_VEL
LIN {X 0,Y 559.184,Z 597.337,A -85,B 0,C 180,E1 -2979.221,E2 -2979.221} C_VEL
LIN {X 0,Y 559.356,Z 587.402,A -85,B 0,C 180,E1 -2980.131,E2 -2980.131} C_VEL
LIN {X 0,Y 559.543,Z 576.403,A -85,B 0,C 180,E1 -2980.937,E2 -2980.937} C_VEL
LIN {X 0,Y 559.671,Z 564.465,A -85,B 0,C 180,E1 -2981.627,E2 -2981.627} C_VEL
LIN {X 0,Y 559.817,Z 551.776,A -85,B 0,C 180,E1 -2982.184,E2 -2982.184} C_VEL
LIN {X 0,Y 559.973,Z 538.358,A -85,B 0,C 180,E1 -2982.595,E2 -2982.595} C_VEL
LIN {X 0,Y 560.106,Z 525.105,A -85,B 0,C 180,E1 -2982.845,E2 -2982.845} C_VEL
LIN {X 0,Y 560.246,Z 428.089,A -85,B 0,C 180,E1 -2984.095,E2 -2984.095} C_VEL
LIN {X 0,Y 559.427,Z 422.441,A -85,B 0,C 180,E1 -2984.203,E2 -2984.203} C_VEL
LIN {X 0,Y 559.682,Z 399.799,A -85,B 0,C 180,E1 -2987.38,E2 -2987.38} C_VEL
LIN {X 0,Y 559.962,Z 379.891,A -85,B 0,C 180,E1 -2990.19,E2 -2990.19} C_VEL
LIN {X 0,Y 560.261,Z 358.187,A -85,B 0,C 180,E1 -2993.274,E2 -2993.274} C_VEL
LIN {X 0,Y 559.191,Z 351.835,A -85,B 0,C 180,E1 -2994.256,E2 -2994.256} C_VEL
LIN {X 0,Y 559.171,Z 351.829,A -85,B 0,C 180,E1 -2996.902,E2 -2996.902} C_VEL
LIN {X 0,Y 559.189,Z 351.832,A -85,B 0,C 180,E1 -2999.864,E2 -2999.864} C_VEL
LIN {X 0,Y 559.175,Z 351.828,A -85,B 0,C 180,E1 -3002.713,E2 -3002.713} C_VEL
LIN {X 0,Y 559.157,Z 351.829,A -85,B 0,C 180,E1 -3005.321,E2 -3005.321} C_VEL
LIN {X 0,Y 559.133,Z 351.84,A -85,B 0,C 180,E1 -3008.017,E2 -3008.017} C_VEL
LIN {X 0,Y 559.174,Z 351.827,A -85,B 0,C 180,E1 -3010.81,E2 -3010.81} C_VEL
LIN {X 0,Y 559.14,Z 351.837,A -85,B 0,C 180,E1 -3013.733,E2 -3013.733} C_VEL
LIN {X 0,Y 559.163,Z 351.828,A -85,B 0,C 180,E1 -3016.8,E2 -3016.8} C_VEL
LIN {X 0,Y 559.172,Z 351.828,A -85,B 0,C 180,E1 -3019.189,E2 -3019.189} C_VEL
LIN {X 0,Y 559.13,Z 351.839,A -85,B 0,C 180,E1 -3021.982,E2 -3021.982} C_VEL
LIN {X 0,Y 559.152,Z 351.829,A -85,B 0,C 180,E1 -3024.782,E2 -3024.782} C_VEL
LIN {X 0,Y 559.168,Z 351.83,A -85,B 0,C 180,E1 -3027.361,E2 -3027.361} C_VEL
LIN {X 0,Y 559.181,Z 351.828,A -85,B 0,C 180,E1 -3030.135,E2 -3030.135} C_VEL
LIN {X 0,Y 559.174,Z 351.828,A -85,B 0,C 180,E1 -3033.169,E2 -3033.169} C_VEL
LIN {X 0,Y 559.148,Z 351.836,A -85,B 0,C 180,E1 -3035.495,E2 -3035.495} C_VEL
LIN {X 0,Y 559.169,Z 351.826,A -85,B 0,C 180,E1 -3038.624,E2 -3038.624} C_VEL
LIN {X 0,Y 559.163,Z 351.829,A -85,B 0,C 180,E1 -3040.926,E2 -3040.926} C_VEL
LIN {X 0,Y 559.164,Z 351.831,A -85,B 0,C 180,E1 -3043.948,E2 -3043.948} C_VEL
LIN {X 0,Y 559.165,Z 351.828,A -85,B 0,C 180,E1 -3046.184,E2 -3046.184} C_VEL
LIN {X 0,Y 559.201,Z 351.827,A -85,B 0,C 180,E1 -3049.134,E2 -3049.134} C_VEL
LIN {X 0,Y 559.202,Z 351.822,A -85,B 0,C 180,E1 -3052.054,E2 -3052.054} C_VEL
LIN {X 0,Y 559.253,Z 351.82,A -85,B 0,C 180,E1 -3054.953,E2 -3054.953} C_VEL
LIN {X 0,Y 559.244,Z 351.819,A -85,B 0,C 180,E1 -3057.84,E2 -3057.84} C_VEL
LIN {X 0,Y 559.27,Z 351.816,A -85,B 0,C 180,E1 -3060.72,E2 -3060.72} C_VEL
LIN {X 0,Y 559.238,Z 351.82,A -85,B 0,C 180,E1 -3062.882,E2 -3062.882} C_VEL
LIN {X 0,Y 559.224,Z 351.822,A -85,B 0,C 180,E1 -3065.77,E2 -3065.77} C_VEL
LIN {X 0,Y 559.197,Z 351.825,A -85,B 0,C 180,E1 -3068.674,E2 -3068.674} C_VEL
LIN {X 0,Y 559.2,Z 351.825,A -85,B 0,C 180,E1 -3071.601,E2 -3071.601} C_VEL
LIN {X 0,Y 559.19,Z 351.827,A -85,B 0,C 180,E1 -3074.596,E2 -3074.596} C_VEL
LIN {X 0,Y 559.157,Z 351.832,A -85,B 0,C 180,E1 -3077.557,E2 -3077.557} C_VEL
LIN {X 0,Y 559.168,Z 351.827,A -85,B 0,C 180,E1 -3079.838,E2 -3079.838} C_VEL
LIN {X 0,Y 559.149,Z 351.83,A -85,B 0,C 180,E1 -3082.153,E2 -3082.153} C_VEL
LIN {X 0,Y 559.153,Z 351.83,A -85,B 0,C 180,E1 -3084.506,E2 -3084.506} C_VEL
LIN {X 0,Y 559.174,Z 351.835,A -85,B 0,C 180,E1 -3086.902,E2 -3086.902} C_VEL
LIN {X 0,Y 559.144,Z 351.83,A -85,B 0,C 180,E1 -3089.859,E2 -3089.859} C_VEL
LIN {X 0,Y 559.141,Z 351.834,A -85,B 0,C 180,E1 -3090.633,E2 -3090.633} C_VEL
LIN {X 0,Y 558.483,Z 351.921,A -85,B 0,C 180,E1 -3091.235,E2 -3091.235} C_VEL
LIN {X 0,Y 555.623,Z 352.275,A -85,B 0,C 180,E1 -3092.211,E2 -3092.211} C_VEL
LIN {X 0,Y 553.211,Z 352.575,A -85,B 0,C 180,E1 -3092.997,E2 -3092.997} C_VEL
LIN {X 0,Y 552.192,Z 352.695,A -85,B 0,C 180,E1 -3093.604,E2 -3093.604} C_VEL
LIN {X 0,Y 552.119,Z 352.703,A -85,B 0,C 180,E1 -3093.809,E2 -3093.809} C_VEL
LIN {X 0,Y 552.108,Z 352.715,A -85,B 0,C 180,E1 -3096.747,E2 -3096.747} C_VEL
LIN {X 0,Y 552.131,Z 352.705,A -85,B 0,C 180,E1 -3099.528,E2 -3099.528} C_VEL
LIN {X 0,Y 552.128,Z 352.708,A -85,B 0,C 180,E1 -3102.426,E2 -3102.426} C_VEL
LIN {X 0,Y 552.098,Z 352.709,A -85,B 0,C 180,E1 -3105.564,E2 -3105.564} C_VEL
LIN {X 0,Y 552.14,Z 352.712,A -85,B 0,C 180,E1 -3108.677,E2 -3108.677} C_VEL
LIN {X 0,Y 552.12,Z 352.709,A -85,B 0,C 180,E1 -3111.412,E2 -3111.412} C_VEL
LIN {X 0,Y 552.111,Z 352.717,A -85,B 0,C 180,E1 -3114.556,E2 -3114.556} C_VEL
LIN {X 0,Y 552.149,Z 352.711,A -85,B 0,C 180,E1 -3115.351,E2 -3115.351} C_VEL
LIN {X 0,Y 552.447,Z 356.792,A -85,B 0,C 180,E1 -3116.182,E2 -3116.182} C_VEL
LIN {X 0,Y 552.186,Z 372.021,A -85,B 0,C 180,E1 -3119.185,E2 -3119.185} C_VEL
LIN {X 0,Y 552.211,Z 374.583,A -85,B 0,C 180,E1 -3119.68,E2 -3119.68} C_VEL
LIN {X 0,Y 553.418,Z 382.986,A -85,B 0,C 180,E1 -3119.836,E2 -3119.836} C_VEL
LIN {X 0,Y 553.104,Z 481.754,A -85,B 0,C 180,E1 -3121.144,E2 -3121.144} C_VEL
LIN {X 0,Y 552.935,Z 495.411,A -85,B 0,C 180,E1 -3121.487,E2 -3121.487} C_VEL
LIN {X 0,Y 552.841,Z 507.618,A -85,B 0,C 180,E1 -3121.943,E2 -3121.943} C_VEL
LIN {X 0,Y 552.625,Z 519.611,A -85,B 0,C 180,E1 -3122.548,E2 -3122.548} C_VEL
LIN {X 0,Y 552.45,Z 530.946,A -85,B 0,C 180,E1 -3123.284,E2 -3123.284} C_VEL
LIN {X 0,Y 552.257,Z 541.73,A -85,B 0,C 180,E1 -3124.16,E2 -3124.16} C_VEL
LIN {X 0,Y 552.075,Z 551.549,A -85,B 0,C 180,E1 -3125.16,E2 -3125.16} C_VEL
LIN {X 0,Y 551.954,Z 560.199,A -85,B 0,C 180,E1 -3126.247,E2 -3126.247} C_VEL
LIN {X 0,Y 551.867,Z 567.203,A -85,B 0,C 180,E1 -3127.342,E2 -3127.342} C_VEL
LIN {X 0,Y 551.791,Z 572.654,A -85,B 0,C 180,E1 -3128.402,E2 -3128.402} C_VEL
LIN {X 0,Y 551.736,Z 577.112,A -85,B 0,C 180,E1 -3129.495,E2 -3129.495} C_VEL
LIN {X 0,Y 551.692,Z 580.68,A -85,B 0,C 180,E1 -3130.658,E2 -3130.658} C_VEL
LIN {X 0,Y 551.65,Z 582.421,A -85,B 0,C 180,E1 -3131.428,E2 -3131.428} C_VEL
LIN {X 0,Y 551.662,Z 584.46,A -85,B 0,C 180,E1 -3132.84,E2 -3132.84} C_VEL
LIN {X 0,Y 551.634,Z 584.937,A -85,B 0,C 180,E1 -3133.723,E2 -3133.723} C_VEL
LIN {X 0,Y 551.607,Z 584.911,A -85,B 0,C 180,E1 -3134.481,E2 -3134.481} C_VEL
LIN {X 0,Y 551.652,Z 584.165,A -85,B 0,C 180,E1 -3135.522,E2 -3135.522} C_VEL
LIN {X 0,Y 551.662,Z 582.256,A -85,B 0,C 180,E1 -3136.744,E2 -3136.744} C_VEL
LIN {X 0,Y 551.734,Z 579.461,A -85,B 0,C 180,E1 -3137.868,E2 -3137.868} C_VEL
LIN {X 0,Y 551.751,Z 575.63,A -85,B 0,C 180,E1 -3138.985,E2 -3138.985} C_VEL
LIN {X 0,Y 551.816,Z 570.66,A -85,B 0,C 180,E1 -3140.1,E2 -3140.1} C_VEL
LIN {X 0,Y 551.882,Z 564.422,A -85,B 0,C 180,E1 -3141.21,E2 -3141.21} C_VEL
LIN {X 0,Y 552.036,Z 556.651,A -85,B 0,C 180,E1 -3142.318,E2 -3142.318} C_VEL
LIN {X 0,Y 552.176,Z 546.965,A -85,B 0,C 180,E1 -3143.422,E2 -3143.422} C_VEL
LIN {X 0,Y 552.313,Z 536.996,A -85,B 0,C 180,E1 -3144.341,E2 -3144.341} C_VEL
LIN {X 0,Y 552.492,Z 525.741,A -85,B 0,C 180,E1 -3145.166,E2 -3145.166} C_VEL
LIN {X 0,Y 552.704,Z 514.728,A -85,B 0,C 180,E1 -3145.807,E2 -3145.807} C_VEL
LIN {X 0,Y 552.886,Z 502.544,A -85,B 0,C 180,E1 -3146.356,E2 -3146.356} C_VEL
LIN {X 0,Y 553.029,Z 489.685,A -85,B 0,C 180,E1 -3146.767,E2 -3146.767} C_VEL
LIN {X 0,Y 553.126,Z 477.495,A -85,B 0,C 180,E1 -3147.018,E2 -3147.018} C_VEL
LIN {X 0,Y 553.286,Z 381.027,A -85,B 0,C 180,E1 -3148.283,E2 -3148.283} C_VEL
LIN {X 0,Y 552.176,Z 374.614,A -85,B 0,C 180,E1 -3148.405,E2 -3148.405} C_VEL
LIN {X 0,Y 552.384,Z 359.1,A -85,B 0,C 180,E1 -3151.458,E2 -3151.458} C_VEL
LIN {X 0,Y 552.323,Z 353.581,A -85,B 0,C 180,E1 -3152.552,E2 -3152.552} C_VEL
LIN {X 0,Y 552.219,Z 352.7,A -85,B 0,C 180,E1 -3152.735,E2 -3152.735} C_VEL
LIN {X 0,Y 552.199,Z 352.7,A -85,B 0,C 180,E1 -3155.844,E2 -3155.844} C_VEL
LIN {X 0,Y 552.152,Z 352.703,A -85,B 0,C 180,E1 -3158.786,E2 -3158.786} C_VEL
LIN {X 0,Y 552.169,Z 352.703,A -85,B 0,C 180,E1 -3161.75,E2 -3161.75} C_VEL
LIN {X 0,Y 552.142,Z 352.704,A -85,B 0,C 180,E1 -3164.748,E2 -3164.748} C_VEL
LIN {X 0,Y 552.114,Z 352.709,A -85,B 0,C 180,E1 -3167.788,E2 -3167.788} C_VEL
LIN {X 0,Y 552.131,Z 352.704,A -85,B 0,C 180,E1 -3170.101,E2 -3170.101} C_VEL
LIN {X 0,Y 552.1,Z 352.708,A -85,B 0,C 180,E1 -3172.45,E2 -3172.45} C_VEL
LIN {X 0,Y 552.159,Z 352.708,A -85,B 0,C 180,E1 -3175.35,E2 -3175.35} C_VEL
LIN {X 0,Y 552.112,Z 352.706,A -85,B 0,C 180,E1 -3178.097,E2 -3178.097} C_VEL
LIN {X 0,Y 552.11,Z 352.708,A -85,B 0,C 180,E1 -3180.608,E2 -3180.608} C_VEL
LIN {X 0,Y 552.125,Z 352.714,A -85,B 0,C 180,E1 -3183.184,E2 -3183.184} C_VEL
LIN {X 0,Y 552.115,Z 352.706,A -85,B 0,C 180,E1 -3185.841,E2 -3185.841} C_VEL
LIN {X 0,Y 552.127,Z 352.714,A -85,B 0,C 180,E1 -3189.061,E2 -3189.061} C_VEL
LIN {X 0,Y 552.139,Z 352.706,A -85,B 0,C 180,E1 -3191.443,E2 -3191.443} C_VEL
LIN {X 0,Y 552.095,Z 352.711,A -85,B 0,C 180,E1 -3194.531,E2 -3194.531} C_VEL
LIN {X 0,Y 552.129,Z 352.706,A -85,B 0,C 180,E1 -3197.583,E2 -3197.583} C_VEL
LIN {X 0,Y 552.131,Z 352.706,A -85,B 0,C 180,E1 -3200.472,E2 -3200.472} C_VEL
LIN {X 0,Y 552.111,Z 352.71,A -85,B 0,C 180,E1 -3203.315,E2 -3203.315} C_VEL
LIN {X 0,Y 552.126,Z 352.704,A -85,B 0,C 180,E1 -3205.939,E2 -3205.939} C_VEL
LIN {X 0,Y 552.113,Z 352.71,A -85,B 0,C 180,E1 -3208.54,E2 -3208.54} C_VEL
LIN {X 0,Y 552.12,Z 352.707,A -85,B 0,C 180,E1 -3211.437,E2 -3211.437} C_VEL
LIN {X 0,Y 552.131,Z 352.707,A -85,B 0,C 180,E1 -3214.355,E2 -3214.355} C_VEL
LIN {X 0,Y 552.104,Z 352.717,A -85,B 0,C 180,E1 -3216.758,E2 -3216.758} C_VEL
LIN {X 0,Y 552.12,Z 352.709,A -85,B 0,C 180,E1 -3219.119,E2 -3219.119} C_VEL
LIN {X 0,Y 552.124,Z 352.705,A -85,B 0,C 180,E1 -3221.444,E2 -3221.444} C_VEL
LIN {X 0,Y 552.114,Z 352.706,A -85,B 0,C 180,E1 -3223.737,E2 -3223.737} C_VEL
LIN {X 0,Y 552.129,Z 352.705,A -85,B 0,C 180,E1 -3226.004,E2 -3226.004} C_VEL
LIN {X 0,Y 552.169,Z 352.703,A -85,B 0,C 180,E1 -3228.993,E2 -3228.993} C_VEL
LIN {X 0,Y 552.155,Z 352.702,A -85,B 0,C 180,E1 -3231.951,E2 -3231.951} C_VEL
LIN {X 0,Y 552.225,Z 352.697,A -85,B 0,C 180,E1 -3234.889,E2 -3234.889} C_VEL
LIN {X 0,Y 552.215,Z 352.694,A -85,B 0,C 180,E1 -3237.812,E2 -3237.812} C_VEL
LIN {X 0,Y 552.238,Z 352.697,A -85,B 0,C 180,E1 -3240.729,E2 -3240.729} C_VEL
LIN {X 0,Y 552.202,Z 352.698,A -85,B 0,C 180,E1 -3242.918,E2 -3242.918} C_VEL
LIN {X 0,Y 552.191,Z 352.697,A -85,B 0,C 180,E1 -3245.844,E2 -3245.844} C_VEL
LIN {X 0,Y 552.162,Z 352.704,A -85,B 0,C 180,E1 -3248.785,E2 -3248.785} C_VEL
LIN {X 0,Y 552.155,Z 352.702,A -85,B 0,C 180,E1 -3251.751,E2 -3251.751} C_VEL
LIN {X 0,Y 552.127,Z 352.708,A -85,B 0,C 180,E1 -3254.749,E2 -3254.749} C_VEL
LIN {X 0,Y 552.107,Z 352.709,A -85,B 0,C 180,E1 -3257.789,E2 -3257.789} C_VEL
LIN {X 0,Y 552.126,Z 352.711,A -85,B 0,C 180,E1 -3260.101,E2 -3260.101} C_VEL
LIN {X 0,Y 552.09,Z 352.716,A -85,B 0,C 180,E1 -3262.451,E2 -3262.451} C_VEL
LIN {X 0,Y 552.148,Z 352.701,A -85,B 0,C 180,E1 -3265.351,E2 -3265.351} C_VEL
LIN {X 0,Y 552.12,Z 352.713,A -85,B 0,C 180,E1 -3268.098,E2 -3268.098} C_VEL
LIN {X 0,Y 552.107,Z 352.71,A -85,B 0,C 180,E1 -3270.609,E2 -3270.609} C_VEL
LIN {X 0,Y 552.122,Z 352.705,A -85,B 0,C 180,E1 -3273.185,E2 -3273.185} C_VEL
LIN {X 0,Y 552.107,Z 352.712,A -85,B 0,C 180,E1 -3275.842,E2 -3275.842} C_VEL
LIN {X 0,Y 552.121,Z 352.705,A -85,B 0,C 180,E1 -3279.063,E2 -3279.063} C_VEL
LIN {X 0,Y 552.135,Z 352.704,A -85,B 0,C 180,E1 -3281.445,E2 -3281.445} C_VEL
LIN {X 0,Y 552.092,Z 352.711,A -85,B 0,C 180,E1 -3284.533,E2 -3284.533} C_VEL
LIN {X 0,Y 552.127,Z 352.708,A -85,B 0,C 180,E1 -3287.585,E2 -3287.585} C_VEL
LIN {X 0,Y 552.133,Z 352.706,A -85,B 0,C 180,E1 -3290.474,E2 -3290.474} C_VEL
LIN {X 0,Y 552.113,Z 352.707,A -85,B 0,C 180,E1 -3293.316,E2 -3293.316} C_VEL
LIN {X 0,Y 552.131,Z 352.713,A -85,B 0,C 180,E1 -3295.94,E2 -3295.94} C_VEL
LIN {X 0,Y 552.118,Z 352.706,A -85,B 0,C 180,E1 -3298.541,E2 -3298.541} C_VEL
LIN {X 0,Y 552.127,Z 352.71,A -85,B 0,C 180,E1 -3301.438,E2 -3301.438} C_VEL
LIN {X 0,Y 552.131,Z 352.71,A -85,B 0,C 180,E1 -3304.356,E2 -3304.356} C_VEL
LIN {X 0,Y 552.186,Z 352.894,A -85,B 0,C 180,E1 -3305.617,E2 -3305.617} C_VEL
LIN {X 0,Y 553.279,Z 358.74,A -85,B 0,C 180,E1 -3306.526,E2 -3306.526} C_VEL
LIN {X 0,Y 553.073,Z 375.561,A -85,B 0,C 180,E1 -3308.963,E2 -3308.963} C_VEL
LIN {X 0,Y 552.739,Z 395.847,A -85,B 0,C 180,E1 -3311.85,E2 -3311.85} C_VEL
LIN {X 0,Y 552.484,Z 414.63,A -85,B 0,C 180,E1 -3314.507,E2 -3314.507} C_VEL
LIN {X 0,Y 552.434,Z 422.524,A -85,B 0,C 180,E1 -3315.625,E2 -3315.625} C_VEL
LIN {X 0,Y 553.449,Z 430.323,A -85,B 0,C 180,E1 -3315.757,E2 -3315.757} C_VEL
LIN {X 0,Y 553.15,Z 530.961,A -85,B 0,C 180,E1 -3317.084,E2 -3317.084} C_VEL
LIN {X 0,Y 552.993,Z 543.465,A -85,B 0,C 180,E1 -3317.383,E2 -3317.383} C_VEL
LIN {X 0,Y 552.835,Z 556.377,A -85,B 0,C 180,E1 -3317.846,E2 -3317.846} C_VEL
LIN {X 0,Y 552.626,Z 568.321,A -85,B 0,C 180,E1 -3318.428,E2 -3318.428} C_VEL
LIN {X 0,Y 552.476,Z 580.199,A -85,B 0,C 180,E1 -3319.186,E2 -3319.186} C_VEL
LIN {X 0,Y 552.299,Z 590.607,A -85,B 0,C 180,E1 -3320.016,E2 -3320.016} C_VEL
LIN {X 0,Y 552.125,Z 599.115,A -85,B 0,C 180,E1 -3320.845,E2 -3320.845} C_VEL
LIN {X 0,Y 552.013,Z 606.962,A -85,B 0,C 180,E1 -3321.765,E2 -3321.765} C_VEL
LIN {X 0,Y 551.889,Z 614.623,A -85,B 0,C 180,E1 -3322.868,E2 -3322.868} C_VEL
LIN {X 0,Y 551.867,Z 621.68,A -85,B 0,C 180,E1 -3324.153,E2 -3324.153} C_VEL
LIN {X 0,Y 551.725,Z 626.373,A -85,B 0,C 180,E1 -3325.251,E2 -3325.251} C_VEL
LIN {X 0,Y 551.75,Z 629.958,A -85,B 0,C 180,E1 -3326.349,E2 -3326.349} C_VEL
LIN {X 0,Y 551.723,Z 631.807,A -85,B 0,C 180,E1 -3327.079,E2 -3327.079} C_VEL
LIN {X 0,Y 551.645,Z 634.184,A -85,B 0,C 180,E1 -3328.54,E2 -3328.54} C_VEL
LIN {X 0,Y 551.64,Z 635,A -85,B 0,C 180,E1 -3330,E2 -3330} C_VEL
LIN {X 0,Y 551.645,Z 634.185,A -85,B 0,C 180,E1 -3331.46,E2 -3331.46} C_VEL
LIN {X 0,Y 551.723,Z 631.81,A -85,B 0,C 180,E1 -3332.921,E2 -3332.921} C_VEL
LIN {X 0,Y 551.763,Z 628.896,A -85,B 0,C 180,E1 -3334.017,E2 -3334.017} C_VEL
LIN {X 0,Y 551.724,Z 624.949,A -85,B 0,C 180,E1 -3335.116,E2 -3335.116} C_VEL
LIN {X 0,Y 551.815,Z 619.124,A -85,B 0,C 180,E1 -3336.353,E2 -3336.353} C_VEL
LIN {X 0,Y 551.926,Z 612.237,A -85,B 0,C 180,E1 -3337.499,E2 -3337.499} C_VEL
LIN {X 0,Y 552.082,Z 603.993,A -85,B 0,C 180,E1 -3338.602,E2 -3338.602} C_VEL
LIN {X 0,Y 552.221,Z 595.542,A -85,B 0,C 180,E1 -3339.523,E2 -3339.523} C_VEL
LIN {X 0,Y 552.432,Z 585.096,A -85,B 0,C 180,E1 -3340.445,E2 -3340.445} C_VEL
LIN {X 0,Y 552.555,Z 574.29,A -85,B 0,C 180,E1 -3341.214,E2 -3341.214} C_VEL
LIN {X 0,Y 552.781,Z 563.411,A -85,B 0,C 180,E1 -3341.83,E2 -3341.83} C_VEL
LIN {X 0,Y 552.884,Z 551.772,A -85,B 0,C 180,E1 -3342.34,E2 -3342.34} C_VEL
LIN {X 0,Y 553.047,Z 538.357,A -85,B 0,C 180,E1 -3342.756,E2 -3342.756} C_VEL
LIN {X 0,Y 553.206,Z 525.105,A -85,B 0,C 180,E1 -3343.009,E2 -3343.009} C_VEL
LIN {X 0,Y 553.393,Z 428.984,A -85,B 0,C 180,E1 -3344.262,E2 -3344.262} C_VEL
LIN {X 0,Y 552.427,Z 422.441,A -85,B 0,C 180,E1 -3344.387,E2 -3344.387} C_VEL
LIN {X 0,Y 552.704,Z 400.385,A -85,B 0,C 180,E1 -3347.507,E2 -3347.507} C_VEL
LIN {X 0,Y 552.974,Z 380.938,A -85,B 0,C 180,E1 -3350.263,E2 -3350.263} C_VEL
LIN {X 0,Y 553.337,Z 360.618,A -85,B 0,C 180,E1 -3353.187,E2 -3353.187} C_VEL
LIN {X 0,Y 552.644,Z 355.193,A -85,B 0,C 180,E1 -3354.012,E2 -3354.012} C_VEL
LIN {X 0,Y 552.157,Z 352.71,A -85,B 0,C 180,E1 -3354.435,E2 -3354.435} C_VEL
LIN {X 0,Y 552.144,Z 352.704,A -85,B 0,C 180,E1 -3357.272,E2 -3357.272} C_VEL
LIN {X 0,Y 552.143,Z 352.711,A -85,B 0,C 180,E1 -3360.055,E2 -3360.055} C_VEL
LIN {X 0,Y 552.128,Z 352.705,A -85,B 0,C 180,E1 -3362.848,E2 -3362.848} C_VEL
LIN {X 0,Y 552.107,Z 352.709,A -85,B 0,C 180,E1 -3365.444,E2 -3365.444} C_VEL
LIN {X 0,Y 552.096,Z 352.717,A -85,B 0,C 180,E1 -3367.885,E2 -3367.885} C_VEL
LIN {X 0,Y 552.14,Z 352.706,A -85,B 0,C 180,E1 -3370.477,E2 -3370.477} C_VEL
LIN {X 0,Y 552.114,Z 352.708,A -85,B 0,C 180,E1 -3373.484,E2 -3373.484} C_VEL
LIN {X 0,Y 552.115,Z 352.707,A -85,B 0,C 180,E1 -3376.577,E2 -3376.577} C_VEL
LIN {X 0,Y 552.137,Z 352.708,A -85,B 0,C 180,E1 -3379.521,E2 -3379.521} C_VEL
LIN {X 0,Y 552.088,Z 352.711,A -85,B 0,C 180,E1 -3382.336,E2 -3382.336} C_VEL
LIN {X 0,Y 552.123,Z 352.706,A -85,B 0,C 180,E1 -3385.054,E2 -3385.054} C_VEL
LIN {X 0,Y 552.121,Z 352.713,A -85,B 0,C 180,E1 -3387.682,E2 -3387.682} C_VEL
LIN {X 0,Y 552.138,Z 352.705,A -85,B 0,C 180,E1 -3390.237,E2 -3390.237} C_VEL
LIN {X 0,Y 552.139,Z 352.703,A -85,B 0,C 180,E1 -3392.997,E2 -3392.997} C_VEL
LIN {X 0,Y 552.105,Z 352.709,A -85,B 0,C 180,E1 -3395.161,E2 -3395.161} C_VEL
LIN {X 0,Y 552.088,Z 352.718,A -85,B 0,C 180,E1 -3397.549,E2 -3397.549} C_VEL
LIN {X 0,Y 552.14,Z 352.703,A -85,B 0,C 180,E1 -3400.373,E2 -3400.373} C_VEL
LIN {X 0,Y 552.149,Z 352.702,A -85,B 0,C 180,E1 -3402.977,E2 -3402.977} C_VEL
LIN {X 0,Y 552.127,Z 352.706,A -85,B 0,C 180,E1 -3406.004,E2 -3406.004} C_VEL
LIN {X 0,Y 552.169,Z 352.701,A -85,B 0,C 180,E1 -3408.994,E2 -3408.994} C_VEL
LIN {X 0,Y 552.155,Z 352.701,A -85,B 0,C 180,E1 -3411.952,E2 -3411.952} C_VEL
LIN {X 0,Y 552.227,Z 352.694,A -85,B 0,C 180,E1 -3414.889,E2 -3414.889} C_VEL
LIN {X 0,Y 552.215,Z 352.695,A -85,B 0,C 180,E1 -3417.812,E2 -3417.812} C_VEL
LIN {X 0,Y 552.239,Z 352.692,A -85,B 0,C 180,E1 -3420.729,E2 -3420.729} C_VEL
LIN {X 0,Y 552.204,Z 352.697,A -85,B 0,C 180,E1 -3422.918,E2 -3422.918} C_VEL
LIN {X 0,Y 552.194,Z 352.697,A -85,B 0,C 180,E1 -3425.844,E2 -3425.844} C_VEL
LIN {X 0,Y 552.164,Z 352.702,A -85,B 0,C 180,E1 -3428.786,E2 -3428.786} C_VEL
LIN {X 0,Y 552.156,Z 352.701,A -85,B 0,C 180,E1 -3431.751,E2 -3431.751} C_VEL
LIN {X 0,Y 552.128,Z 352.708,A -85,B 0,C 180,E1 -3434.749,E2 -3434.749} C_VEL
LIN {X 0,Y 552.108,Z 352.708,A -85,B 0,C 180,E1 -3437.789,E2 -3437.789} C_VEL
LIN {X 0,Y 552.127,Z 352.703,A -85,B 0,C 180,E1 -3440.102,E2 -3440.102} C_VEL
LIN {X 0,Y 552.108,Z 352.709,A -85,B 0,C 180,E1 -3442.451,E2 -3442.451} C_VEL
LIN {X 0,Y 552.15,Z 352.706,A -85,B 0,C 180,E1 -3445.352,E2 -3445.352} C_VEL
LIN {X 0,Y 552.121,Z 352.705,A -85,B 0,C 180,E1 -3448.098,E2 -3448.098} C_VEL
LIN {X 0,Y 552.102,Z 352.712,A -85,B 0,C 180,E1 -3450.629,E2 -3450.629} C_VEL
LIN {X 0,Y 552.124,Z 352.707,A -85,B 0,C 180,E1 -3453.186,E2 -3453.186} C_VEL
LIN {X 0,Y 552.119,Z 352.703,A -85,B 0,C 180,E1 -3453.809,E2 -3453.809} C_VEL
LIN {X 0,Y 551.484,Z 352.786,A -85,B 0,C 180,E1 -3454.418,E2 -3454.418} C_VEL
LIN {X 0,Y 548.658,Z 353.146,A -85,B 0,C 180,E1 -3455.406,E2 -3455.406} C_VEL
LIN {X 0,Y 546.233,Z 353.452,A -85,B 0,C 180,E1 -3456.201,E2 -3456.201} C_VEL
LIN {X 0,Y 545.162,Z 353.582,A -85,B 0,C 180,E1 -3456.815,E2 -3456.815} C_VEL
LIN {X 0,Y 545.06,Z 353.591,A -85,B 0,C 180,E1 -3457.023,E2 -3457.023} C_VEL
LIN {X 0,Y 545.071,Z 353.584,A -85,B 0,C 180,E1 -3460.143,E2 -3460.143} C_VEL
LIN {X 0,Y 545.086,Z 353.587,A -85,B 0,C 180,E1 -3463.107,E2 -3463.107} C_VEL
LIN {X 0,Y 545.063,Z 353.588,A -85,B 0,C 180,E1 -3466.225,E2 -3466.225} C_VEL
LIN {X 0,Y 545.097,Z 353.588,A -85,B 0,C 180,E1 -3468.888,E2 -3468.888} C_VEL
LIN {X 0,Y 545.054,Z 353.589,A -85,B 0,C 180,E1 -3471.764,E2 -3471.764} C_VEL
LIN {X 0,Y 545.068,Z 353.594,A -85,B 0,C 180,E1 -3474.535,E2 -3474.535} C_VEL
LIN {X 0,Y 545.133,Z 353.691,A -85,B 0,C 180,E1 -3475.245,E2 -3475.245} C_VEL
LIN {X 0,Y 545.509,Z 357.171,A -85,B 0,C 180,E1 -3475.967,E2 -3475.967} C_VEL
LIN {X 0,Y 545.197,Z 373.197,A -85,B 0,C 180,E1 -3479.17,E2 -3479.17} C_VEL
LIN {X 0,Y 545.223,Z 375.119,A -85,B 0,C 180,E1 -3479.51,E2 -3479.51} C_VEL
LIN {X 0,Y 546.555,Z 382.791,A -85,B 0,C 180,E1 -3479.649,E2 -3479.649} C_VEL
LIN {X 0,Y 546.225,Z 481.203,A -85,B 0,C 180,E1 -3480.965,E2 -3480.965} C_VEL
LIN {X 0,Y 546.031,Z 494.508,A -85,B 0,C 180,E1 -3481.296,E2 -3481.296} C_VEL
LIN {X 0,Y 545.866,Z 507.071,A -85,B 0,C 180,E1 -3481.761,E2 -3481.761} C_VEL
LIN {X 0,Y 545.656,Z 519.215,A -85,B 0,C 180,E1 -3482.376,E2 -3482.376} C_VEL
LIN {X 0,Y 545.482,Z 529.693,A -85,B 0,C 180,E1 -3483.053,E2 -3483.053} C_VEL
LIN {X 0,Y 545.255,Z 540.33,A -85,B 0,C 180,E1 -3483.906,E2 -3483.906} C_VEL
LIN {X 0,Y 545.088,Z 549.575,A -85,B 0,C 180,E1 -3484.82,E2 -3484.82} C_VEL
LIN {X 0,Y 544.942,Z 557.826,A -85,B 0,C 180,E1 -3485.819,E2 -3485.819} C_VEL
LIN {X 0,Y 544.797,Z 565.894,A -85,B 0,C 180,E1 -3487.032,E2 -3487.032} C_VEL
LIN {X 0,Y 544.703,Z 572.429,A -85,B 0,C 180,E1 -3488.277,E2 -3488.277} C_VEL
LIN {X 0,Y 544.656,Z 577.699,A -85,B 0,C 180,E1 -3489.611,E2 -3489.611} C_VEL
LIN {X 0,Y 544.616,Z 580.107,A -85,B 0,C 180,E1 -3490.397,E2 -3490.397} C_VEL
LIN {X 0,Y 544.558,Z 581.995,A -85,B 0,C 180,E1 -3491.177,E2 -3491.177} C_VEL
LIN {X 0,Y 544.555,Z 583.395,A -85,B 0,C 180,E1 -3491.957,E2 -3491.957} C_VEL
LIN {X 0,Y 544.582,Z 584.379,A -85,B 0,C 180,E1 -3492.747,E2 -3492.747} C_VEL
LIN {X 0,Y 544.558,Z 584.89,A -85,B 0,C 180,E1 -3493.506,E2 -3493.506} C_VEL
LIN {X 0,Y 544.531,Z 584.957,A -85,B 0,C 180,E1 -3494.274,E2 -3494.274} C_VEL
LIN {X 0,Y 544.56,Z 584.258,A -85,B 0,C 180,E1 -3495.454,E2 -3495.454} C_VEL
LIN {X 0,Y 544.559,Z 582.669,A -85,B 0,C 180,E1 -3496.567,E2 -3496.567} C_VEL
LIN {X 0,Y 544.629,Z 580.066,A -85,B 0,C 180,E1 -3497.707,E2 -3497.707} C_VEL
LIN {X 0,Y 544.669,Z 576.434,A -85,B 0,C 180,E1 -3498.84,E2 -3498.84} C_VEL
LIN {X 0,Y 544.707,Z 571.681,A -85,B 0,C 180,E1 -3499.969,E2 -3499.969} C_VEL
LIN {X 0,Y 544.818,Z 564.55,A -85,B 0,C 180,E1 -3501.282,E2 -3501.282} C_VEL
LIN {X 0,Y 544.975,Z 556.823,A -85,B 0,C 180,E1 -3502.404,E2 -3502.404} C_VEL
LIN {X 0,Y 545.125,Z 547.173,A -85,B 0,C 180,E1 -3503.523,E2 -3503.523} C_VEL
LIN {X 0,Y 545.294,Z 537.25,A -85,B 0,C 180,E1 -3504.453,E2 -3504.453} C_VEL
LIN {X 0,Y 545.519,Z 526.054,A -85,B 0,C 180,E1 -3505.289,E2 -3505.289} C_VEL
LIN {X 0,Y 545.757,Z 515.11,A -85,B 0,C 180,E1 -3505.939,E2 -3505.939} C_VEL
LIN {X 0,Y 545.941,Z 503.079,A -85,B 0,C 180,E1 -3506.494,E2 -3506.494} C_VEL
LIN {X 0,Y 546.121,Z 490.514,A -85,B 0,C 180,E1 -3506.911,E2 -3506.911} C_VEL
LIN {X 0,Y 546.213,Z 478.855,A -85,B 0,C 180,E1 -3507.165,E2 -3507.165} C_VEL
LIN {X 0,Y 546.409,Z 381.852,A -85,B 0,C 180,E1 -3508.457,E2 -3508.457} C_VEL
LIN {X 0,Y 545.139,Z 374.878,A -85,B 0,C 180,E1 -3508.592,E2 -3508.592} C_VEL
LIN {X 0,Y 545.401,Z 360.383,A -85,B 0,C 180,E1 -3511.477,E2 -3511.477} C_VEL
LIN {X 0,Y 545.351,Z 354.851,A -85,B 0,C 180,E1 -3512.585,E2 -3512.585} C_VEL
LIN {X 0,Y 545.191,Z 353.576,A -85,B 0,C 180,E1 -3512.863,E2 -3512.863} C_VEL
LIN {X 0,Y 545.169,Z 353.575,A -85,B 0,C 180,E1 -3515.919,E2 -3515.919} C_VEL
LIN {X 0,Y 545.114,Z 353.581,A -85,B 0,C 180,E1 -3518.9,E2 -3518.9} C_VEL
LIN {X 0,Y 545.141,Z 353.577,A -85,B 0,C 180,E1 -3521.904,E2 -3521.904} C_VEL
LIN {X 0,Y 545.091,Z 353.584,A -85,B 0,C 180,E1 -3524.943,E2 -3524.943} C_VEL
LIN {X 0,Y 545.082,Z 353.582,A -85,B 0,C 180,E1 -3528.025,E2 -3528.025} C_VEL
LIN {X 0,Y 545.097,Z 353.58,A -85,B 0,C 180,E1 -3530.372,E2 -3530.372} C_VEL
LIN {X 0,Y 545.096,Z 353.585,A -85,B 0,C 180,E1 -3533.558,E2 -3533.558} C_VEL
LIN {X 0,Y 545.083,Z 353.582,A -85,B 0,C 180,E1 -3536,E2 -3536} C_VEL
LIN {X 0,Y 545.092,Z 353.583,A -85,B 0,C 180,E1 -3538.747,E2 -3538.747} C_VEL
LIN {X 0,Y 545.08,Z 353.584,A -85,B 0,C 180,E1 -3541.682,E2 -3541.682} C_VEL
LIN {X 0,Y 545.083,Z 353.583,A -85,B 0,C 180,E1 -3544.562,E2 -3544.562} C_VEL
LIN {X 0,Y 545.041,Z 353.593,A -85,B 0,C 180,E1 -3547.303,E2 -3547.303} C_VEL
LIN {X 0,Y 545.074,Z 353.583,A -85,B 0,C 180,E1 -3550.141,E2 -3550.141} C_VEL
LIN {X 0,Y 545.062,Z 353.588,A -85,B 0,C 180,E1 -3552.696,E2 -3552.696} C_VEL
LIN {X 0,Y 545.061,Z 353.592,A -85,B 0,C 180,E1 -3555.166,E2 -3555.166} C_VEL
LIN {X 0,Y 545.081,Z 353.582,A -85,B 0,C 180,E1 -3557.897,E2 -3557.897} C_VEL
LIN {X 0,Y 545.081,Z 353.589,A -85,B 0,C 180,E1 -3560.818,E2 -3560.818} C_VEL
LIN {X 0,Y 545.051,Z 353.586,A -85,B 0,C 180,E1 -3563.62,E2 -3563.62} C_VEL
LIN {X 0,Y 545.066,Z 353.585,A -85,B 0,C 180,E1 -3566.328,E2 -3566.328} C_VEL
LIN {X 0,Y 545.062,Z 353.593,A -85,B 0,C 180,E1 -3568.951,E2 -3568.951} C_VEL
LIN {X 0,Y 545.098,Z 353.581,A -85,B 0,C 180,E1 -3571.507,E2 -3571.507} C_VEL
LIN {X 0,Y 545.093,Z 353.585,A -85,B 0,C 180,E1 -3574.489,E2 -3574.489} C_VEL
LIN {X 0,Y 545.039,Z 353.59,A -85,B 0,C 180,E1 -3577.242,E2 -3577.242} C_VEL
LIN {X 0,Y 545.113,Z 353.582,A -85,B 0,C 180,E1 -3580.414,E2 -3580.414} C_VEL
LIN {X 0,Y 545.07,Z 353.583,A -85,B 0,C 180,E1 -3583.521,E2 -3583.521} C_VEL
LIN {X 0,Y 545.087,Z 353.581,A -85,B 0,C 180,E1 -3585.819,E2 -3585.819} C_VEL
LIN {X 0,Y 545.124,Z 353.583,A -85,B 0,C 180,E1 -3588.849,E2 -3588.849} C_VEL
LIN {X 0,Y 545.126,Z 353.577,A -85,B 0,C 180,E1 -3591.847,E2 -3591.847} C_VEL
LIN {X 0,Y 545.2,Z 353.573,A -85,B 0,C 180,E1 -3594.823,E2 -3594.823} C_VEL
LIN {X 0,Y 545.187,Z 353.569,A -85,B 0,C 180,E1 -3597.783,E2 -3597.783} C_VEL
LIN {X 0,Y 545.207,Z 353.572,A -85,B 0,C 180,E1 -3600.738,E2 -3600.738} C_VEL
LIN {X 0,Y 545.168,Z 353.574,A -85,B 0,C 180,E1 -3602.956,E2 -3602.956} C_VEL
LIN {X 0,Y 545.163,Z 353.574,A -85,B 0,C 180,E1 -3605.919,E2 -3605.919} C_VEL
LIN {X 0,Y 545.119,Z 353.58,A -85,B 0,C 180,E1 -3608.9,E2 -3608.9} C_VEL
LIN {X 0,Y 545.126,Z 353.579,A -85,B 0,C 180,E1 -3611.904,E2 -3611.904} C_VEL
LIN {X 0,Y 545.076,Z 353.584,A -85,B 0,C 180,E1 -3614.944,E2 -3614.944} C_VEL
LIN {X 0,Y 545.075,Z 353.587,A -85,B 0,C 180,E1 -3618.026,E2 -3618.026} C_VEL
LIN {X 0,Y 545.09,Z 353.589,A -85,B 0,C 180,E1 -3620.372,E2 -3620.372} C_VEL
LIN {X 0,Y 545.084,Z 353.582,A -85,B 0,C 180,E1 -3623.559,E2 -3623.559} C_VEL
LIN {X 0,Y 545.081,Z 353.588,A -85,B 0,C 180,E1 -3626,E2 -3626} C_VEL
LIN {X 0,Y 545.085,Z 353.583,A -85,B 0,C 180,E1 -3628.75,E2 -3628.75} C_VEL
LIN {X 0,Y 545.071,Z 353.586,A -85,B 0,C 180,E1 -3631.683,E2 -3631.683} C_VEL
LIN {X 0,Y 545.078,Z 353.585,A -85,B 0,C 180,E1 -3634.563,E2 -3634.563} C_VEL
LIN {X 0,Y 545.034,Z 353.588,A -85,B 0,C 180,E1 -3637.304,E2 -3637.304} C_VEL
LIN {X 0,Y 545.088,Z 353.59,A -85,B 0,C 180,E1 -3640.141,E2 -3640.141} C_VEL
LIN {X 0,Y 545.082,Z 353.582,A -85,B 0,C 180,E1 -3643.106,E2 -3643.106} C_VEL
LIN {X 0,Y 545.063,Z 353.59,A -85,B 0,C 180,E1 -3646.225,E2 -3646.225} C_VEL
LIN {X 0,Y 545.098,Z 353.58,A -85,B 0,C 180,E1 -3648.888,E2 -3648.888} C_VEL
LIN {X 0,Y 545.053,Z 353.592,A -85,B 0,C 180,E1 -3651.764,E2 -3651.764} C_VEL
LIN {X 0,Y 545.064,Z 353.585,A -85,B 0,C 180,E1 -3654.535,E2 -3654.535} C_VEL
LIN {X 0,Y 545.081,Z 353.583,A -85,B 0,C 180,E1 -3657.213,E2 -3657.213} C_VEL
LIN {X 0,Y 545.102,Z 353.588,A -85,B 0,C 180,E1 -3659.814,E2 -3659.814} C_VEL
LIN {X 0,Y 545.097,Z 353.583,A -85,B 0,C 180,E1 -3662.827,E2 -3662.827} C_VEL
LIN {X 0,Y 545.108,Z 353.652,A -85,B 0,C 180,E1 -3665.431,E2 -3665.431} C_VEL
LIN {X 0,Y 546.369,Z 360.436,A -85,B 0,C 180,E1 -3666.5,E2 -3666.5} C_VEL
LIN {X 0,Y 546.086,Z 377.987,A -85,B 0,C 180,E1 -3669.076,E2 -3669.076} C_VEL
LIN {X 0,Y 545.742,Z 398.27,A -85,B 0,C 180,E1 -3671.997,E2 -3671.997} C_VEL
LIN {X 0,Y 545.424,Z 420.131,A -85,B 0,C 180,E1 -3675.107,E2 -3675.107} C_VEL
LIN {X 0,Y 545.443,Z 422.687,A -85,B 0,C 180,E1 -3675.444,E2 -3675.444} C_VEL
LIN {X 0,Y 546.578,Z 430.525,A -85,B 0,C 180,E1 -3675.578,E2 -3675.578} C_VEL
LIN {X 0,Y 546.254,Z 530.961,A -85,B 0,C 180,E1 -3676.918,E2 -3676.918} C_VEL
LIN {X 0,Y 546.061,Z 544.226,A -85,B 0,C 180,E1 -3677.244,E2 -3677.244} C_VEL
LIN {X 0,Y 545.891,Z 556.375,A -85,B 0,C 180,E1 -3677.688,E2 -3677.688} C_VEL
LIN {X 0,Y 545.699,Z 567.471,A -85,B 0,C 180,E1 -3678.231,E2 -3678.231} C_VEL
LIN {X 0,Y 545.525,Z 578.906,A -85,B 0,C 180,E1 -3678.952,E2 -3678.952} C_VEL
LIN {X 0,Y 545.286,Z 589.539,A -85,B 0,C 180,E1 -3679.792,E2 -3679.792} C_VEL
LIN {X 0,Y 545.084,Z 599.115,A -85,B 0,C 180,E1 -3680.726,E2 -3680.726} C_VEL
LIN {X 0,Y 544.977,Z 606.962,A -85,B 0,C 180,E1 -3681.658,E2 -3681.658} C_VEL
LIN {X 0,Y 544.823,Z 614.622,A -85,B 0,C 180,E1 -3682.775,E2 -3682.775} C_VEL
LIN {X 0,Y 544.776,Z 621.68,A -85,B 0,C 180,E1 -3684.076,E2 -3684.076} C_VEL
LIN {X 0,Y 544.629,Z 626.373,A -85,B 0,C 180,E1 -3685.189,E2 -3685.189} C_VEL
LIN {X 0,Y 544.669,Z 629.958,A -85,B 0,C 180,E1 -3686.301,E2 -3686.301} C_VEL
LIN {X 0,Y 544.65,Z 631.807,A -85,B 0,C 180,E1 -3687.041,E2 -3687.041} C_VEL
LIN {X 0,Y 544.546,Z 634.183,A -85,B 0,C 180,E1 -3688.521,E2 -3688.521} C_VEL
LIN {X 0,Y 544.541,Z 635,A -85,B 0,C 180,E1 -3690,E2 -3690} C_VEL
LIN {X 0,Y 544.546,Z 634.184,A -85,B 0,C 180,E1 -3691.479,E2 -3691.479} C_VEL
LIN {X 0,Y 544.65,Z 631.81,A -85,B 0,C 180,E1 -3692.959,E2 -3692.959} C_VEL
LIN {X 0,Y 544.683,Z 628.896,A -85,B 0,C 180,E1 -3694.069,E2 -3694.069} C_VEL
LIN {X 0,Y 544.654,Z 624.949,A -85,B 0,C 180,E1 -3695.182,E2 -3695.182} C_VEL
LIN {X 0,Y 544.729,Z 619.643,A -85,B 0,C 180,E1 -3696.34,E2 -3696.34} C_VEL
LIN {X 0,Y 544.836,Z 613.468,A -85,B 0,C 180,E1 -3697.411,E2 -3697.411} C_VEL
LIN {X 0,Y 545.006,Z 605.479,A -85,B 0,C 180,E1 -3698.528,E2 -3698.528} C_VEL
LIN {X 0,Y 545.152,Z 597.335,A -85,B 0,C 180,E1 -3699.46,E2 -3699.46} C_VEL
LIN {X 0,Y 545.376,Z 587.4,A -85,B 0,C 180,E1 -3700.393,E2 -3700.393} C_VEL
LIN {X 0,Y 545.569,Z 576.596,A -85,B 0,C 180,E1 -3701.207,E2 -3701.207} C_VEL
LIN {X 0,Y 545.746,Z 565.176,A -85,B 0,C 180,E1 -3701.89,E2 -3701.89} C_VEL
LIN {X 0,Y 545.93,Z 552.979,A -85,B 0,C 180,E1 -3702.452,E2 -3702.452} C_VEL
LIN {X 0,Y 546.121,Z 540.184,A -85,B 0,C 180,E1 -3702.873,E2 -3702.873} C_VEL
LIN {X 0,Y 546.297,Z 526.619,A -85,B 0,C 180,E1 -3703.152,E2 -3703.152} C_VEL
LIN {X 0,Y 546.456,Z 429.557,A -85,B 0,C 180,E1 -3704.438,E2 -3704.438} C_VEL
LIN {X 0,Y 545.439,Z 422.47,A -85,B 0,C 180,E1 -3704.561,E2 -3704.561} C_VEL
LIN {X 0,Y 545.696,Z 399.955,A -85,B 0,C 180,E1 -3707.757,E2 -3707.757} C_VEL
LIN {X 0,Y 546.053,Z 379.275,A -85,B 0,C 180,E1 -3710.728,E2 -3710.728} C_VEL
LIN {X 0,Y 546.362,Z 360.35,A -85,B 0,C 180,E1 -3713.5,E2 -3713.5} C_VEL
LIN {X 0,Y 545.108,Z 353.586,A -85,B 0,C 180,E1 -3714.569,E2 -3714.569} C_VEL
LIN {X 0,Y 545.094,Z 353.585,A -85,B 0,C 180,E1 -3717.655,E2 -3717.655} C_VEL
LIN {X 0,Y 545.096,Z 353.589,A -85,B 0,C 180,E1 -3720.249,E2 -3720.249} C_VEL
LIN {X 0,Y 545.088,Z 353.581,A -85,B 0,C 180,E1 -3723.063,E2 -3723.063} C_VEL
LIN {X 0,Y 545.062,Z 353.589,A -85,B 0,C 180,E1 -3725.677,E2 -3725.677} C_VEL
LIN {X 0,Y 545.052,Z 353.591,A -85,B 0,C 180,E1 -3728.236,E2 -3728.236} C_VEL
LIN {X 0,Y 545.098,Z 353.581,A -85,B 0,C 180,E1 -3731.112,E2 -3731.112} C_VEL
LIN {X 0,Y 545.055,Z 353.592,A -85,B 0,C 180,E1 -3734.128,E2 -3734.128} C_VEL
LIN {X 0,Y 545.082,Z 353.582,A -85,B 0,C 180,E1 -3736.894,E2 -3736.894} C_VEL
LIN {X 0,Y 545.088,Z 353.59,A -85,B 0,C 180,E1 -3739.859,E2 -3739.859} C_VEL
LIN {X 0,Y 545.069,Z 353.584,A -85,B 0,C 180,E1 -3743.072,E2 -3743.072} C_VEL
LIN {X 0,Y 545.083,Z 353.589,A -85,B 0,C 180,E1 -3745.605,E2 -3745.605} C_VEL
LIN {X 0,Y 545.071,Z 353.585,A -85,B 0,C 180,E1 -3748.317,E2 -3748.317} C_VEL
LIN {X 0,Y 545.085,Z 353.584,A -85,B 0,C 180,E1 -3751.25,E2 -3751.25} C_VEL
LIN {X 0,Y 545.081,Z 353.586,A -85,B 0,C 180,E1 -3754,E2 -3754} C_VEL
LIN {X 0,Y 545.082,Z 353.582,A -85,B 0,C 180,E1 -3756.441,E2 -3756.441} C_VEL
LIN {X 0,Y 545.09,Z 353.59,A -85,B 0,C 180,E1 -3759.628,E2 -3759.628} C_VEL
LIN {X 0,Y 545.087,Z 353.58,A -85,B 0,C 180,E1 -3762.75,E2 -3762.75} C_VEL
LIN {X 0,Y 545.086,Z 353.586,A -85,B 0,C 180,E1 -3765.82,E2 -3765.82} C_VEL
LIN {X 0,Y 545.123,Z 353.577,A -85,B 0,C 180,E1 -3768.85,E2 -3768.85} C_VEL
LIN {X 0,Y 545.126,Z 353.577,A -85,B 0,C 180,E1 -3771.847,E2 -3771.847} C_VEL
LIN {X 0,Y 545.202,Z 353.569,A -85,B 0,C 180,E1 -3774.823,E2 -3774.823} C_VEL
LIN {X 0,Y 545.187,Z 353.571,A -85,B 0,C 180,E1 -3777.784,E2 -3777.784} C_VEL
LIN {X 0,Y 545.209,Z 353.568,A -85,B 0,C 180,E1 -3780.739,E2 -3780.739} C_VEL
LIN {X 0,Y 545.17,Z 353.573,A -85,B 0,C 180,E1 -3782.956,E2 -3782.956} C_VEL
LIN {X 0,Y 545.165,Z 353.572,A -85,B 0,C 180,E1 -3785.92,E2 -3785.92} C_VEL
LIN {X 0,Y 545.121,Z 353.581,A -85,B 0,C 180,E1 -3788.9,E2 -3788.9} C_VEL
LIN {X 0,Y 545.127,Z 353.575,A -85,B 0,C 180,E1 -3791.905,E2 -3791.905} C_VEL
LIN {X 0,Y 545.078,Z 353.589,A -85,B 0,C 180,E1 -3794.944,E2 -3794.944} C_VEL
LIN {X 0,Y 545.077,Z 353.583,A -85,B 0,C 180,E1 -3798.026,E2 -3798.026} C_VEL
LIN {X 0,Y 545.092,Z 353.58,A -85,B 0,C 180,E1 -3800.373,E2 -3800.373} C_VEL
LIN {X 0,Y 545.107,Z 353.579,A -85,B 0,C 180,E1 -3803.558,E2 -3803.558} C_VEL
LIN {X 0,Y 545.083,Z 353.582,A -85,B 0,C 180,E1 -3806.001,E2 -3806.001} C_VEL
LIN {X 0,Y 545.085,Z 353.588,A -85,B 0,C 180,E1 -3808.75,E2 -3808.75} C_VEL
LIN {X 0,Y 545.073,Z 353.584,A -85,B 0,C 180,E1 -3811.683,E2 -3811.683} C_VEL
LIN {X 0,Y 545.08,Z 353.585,A -85,B 0,C 180,E1 -3814.564,E2 -3814.564} C_VEL
LIN {X 0,Y 545.06,Z 353.591,A -85,B 0,C 180,E1 -3817.023,E2 -3817.023} C_VEL
LIN {X 0,Y 544.352,Z 353.676,A -85,B 0,C 180,E1 -3817.639,E2 -3817.639} C_VEL
LIN {X 0,Y 541.485,Z 354.037,A -85,B 0,C 180,E1 -3818.64,E2 -3818.64} C_VEL
LIN {X 0,Y 539.102,Z 354.329,A -85,B 0,C 180,E1 -3819.446,E2 -3819.446} C_VEL
LIN {X 0,Y 538.102,Z 354.452,A -85,B 0,C 180,E1 -3820.068,E2 -3820.068} C_VEL
LIN {X 0,Y 538.032,Z 354.463,A -85,B 0,C 180,E1 -3820.278,E2 -3820.278} C_VEL
LIN {X 0,Y 538.032,Z 354.467,A -85,B 0,C 180,E1 -3822.99,E2 -3822.99} C_VEL
LIN {X 0,Y 538.027,Z 354.462,A -85,B 0,C 180,E1 -3825.926,E2 -3825.926} C_VEL
LIN {X 0,Y 538.051,Z 354.462,A -85,B 0,C 180,E1 -3829.226,E2 -3829.226} C_VEL
LIN {X 0,Y 537.995,Z 354.471,A -85,B 0,C 180,E1 -3832.123,E2 -3832.123} C_VEL
LIN {X 0,Y 538.094,Z 354.508,A -85,B 0,C 180,E1 -3835.108,E2 -3835.108} C_VEL
LIN {X 0,Y 538.502,Z 359.216,A -85,B 0,C 180,E1 -3836.086,E2 -3836.086} C_VEL
LIN {X 0,Y 538.216,Z 375.279,A -85,B 0,C 180,E1 -3839.314,E2 -3839.314} C_VEL
LIN {X 0,Y 539.685,Z 384.339,A -85,B 0,C 180,E1 -3839.478,E2 -3839.478} C_VEL
LIN {X 0,Y 539.33,Z 481.598,A -85,B 0,C 180,E1 -3840.797,E2 -3840.797} C_VEL
LIN {X 0,Y 539.116,Z 495.017,A -85,B 0,C 180,E1 -3841.136,E2 -3841.136} C_VEL
LIN {X 0,Y 538.951,Z 508.075,A -85,B 0,C 180,E1 -3841.632,E2 -3841.632} C_VEL
LIN {X 0,Y 538.72,Z 519.595,A -85,B 0,C 180,E1 -3842.229,E2 -3842.229} C_VEL
LIN {X 0,Y 538.465,Z 531.572,A -85,B 0,C 180,E1 -3843.029,E2 -3843.029} C_VEL
LIN {X 0,Y 538.247,Z 541.193,A -85,B 0,C 180,E1 -3843.832,E2 -3843.832} C_VEL
LIN {X 0,Y 538.082,Z 549.512,A -85,B 0,C 180,E1 -3844.676,E2 -3844.676} C_VEL
LIN {X 0,Y 537.908,Z 557.82,A -85,B 0,C 180,E1 -3845.698,E2 -3845.698} C_VEL
LIN {X 0,Y 537.725,Z 565.782,A -85,B 0,C 180,E1 -3846.916,E2 -3846.916} C_VEL
LIN {X 0,Y 537.649,Z 572.151,A -85,B 0,C 180,E1 -3848.141,E2 -3848.141} C_VEL
LIN {X 0,Y 537.585,Z 576.964,A -85,B 0,C 180,E1 -3849.331,E2 -3849.331} C_VEL
LIN {X 0,Y 537.522,Z 579.934,A -85,B 0,C 180,E1 -3850.287,E2 -3850.287} C_VEL
LIN {X 0,Y 537.451,Z 583.065,A -85,B 0,C 180,E1 -3851.71,E2 -3851.71} C_VEL
LIN {X 0,Y 537.472,Z 584.306,A -85,B 0,C 180,E1 -3852.661,E2 -3852.661} C_VEL
LIN {X 0,Y 537.43,Z 585,A -85,B 0,C 180,E1 -3854.061,E2 -3854.061} C_VEL
LIN {X 0,Y 537.477,Z 584.355,A -85,B 0,C 180,E1 -3855.381,E2 -3855.381} C_VEL
LIN {X 0,Y 537.473,Z 583.052,A -85,B 0,C 180,E1 -3856.387,E2 -3856.387} C_VEL
LIN {X 0,Y 537.493,Z 581.543,A -85,B 0,C 180,E1 -3857.157,E2 -3857.157} C_VEL
LIN {X 0,Y 537.551,Z 578.454,A -85,B 0,C 180,E1 -3858.309,E2 -3858.309} C_VEL
LIN {X 0,Y 537.583,Z 574.299,A -85,B 0,C 180,E1 -3859.454,E2 -3859.454} C_VEL
LIN {X 0,Y 537.691,Z 567.951,A -85,B 0,C 180,E1 -3860.787,E2 -3860.787} C_VEL
LIN {X 0,Y 537.839,Z 561.105,A -85,B 0,C 180,E1 -3861.925,E2 -3861.925} C_VEL
LIN {X 0,Y 537.987,Z 553.122,A -85,B 0,C 180,E1 -3862.995,E2 -3862.995} C_VEL
LIN {X 0,Y 538.15,Z 543.84,A -85,B 0,C 180,E1 -3864.003,E2 -3864.003} C_VEL
LIN {X 0,Y 538.411,Z 533.1,A -85,B 0,C 180,E1 -3864.945,E2 -3864.945} C_VEL
LIN {X 0,Y 538.609,Z 522.332,A -85,B 0,C 180,E1 -3865.697,E2 -3865.697} C_VEL
LIN {X 0,Y 538.911,Z 510.239,A -85,B 0,C 180,E1 -3866.355,E2 -3866.355} C_VEL
LIN {X 0,Y 539.092,Z 497.634,A -85,B 0,C 180,E1 -3866.871,E2 -3866.871} C_VEL
LIN {X 0,Y 539.22,Z 485.071,A -85,B 0,C 180,E1 -3867.222,E2 -3867.222} C_VEL
LIN {X 0,Y 539.396,Z 467.211,A -85,B 0,C 180,E1 -3867.503,E2 -3867.503} C_VEL
LIN {X 0,Y 539.564,Z 382.732,A -85,B 0,C 180,E1 -3868.636,E2 -3868.636} C_VEL
LIN {X 0,Y 538.132,Z 375.172,A -85,B 0,C 180,E1 -3868.784,E2 -3868.784} C_VEL
LIN {X 0,Y 538.413,Z 361.69,A -85,B 0,C 180,E1 -3871.496,E2 -3871.496} C_VEL
LIN {X 0,Y 538.376,Z 356.138,A -85,B 0,C 180,E1 -3872.619,E2 -3872.619} C_VEL
LIN {X 0,Y 538.144,Z 354.455,A -85,B 0,C 180,E1 -3872.994,E2 -3872.994} C_VEL
LIN {X 0,Y 538.12,Z 354.453,A -85,B 0,C 180,E1 -3875.997,E2 -3875.997} C_VEL
LIN {X 0,Y 538.067,Z 354.46,A -85,B 0,C 180,E1 -3879.017,E2 -3879.017} C_VEL
LIN {X 0,Y 538.09,Z 354.454,A -85,B 0,C 180,E1 -3882.062,E2 -3882.062} C_VEL
LIN {X 0,Y 538.05,Z 354.464,A -85,B 0,C 180,E1 -3885.143,E2 -3885.143} C_VEL
LIN {X 0,Y 538.034,Z 354.46,A -85,B 0,C 180,E1 -3888.27,E2 -3888.27} C_VEL
LIN {X 0,Y 538.042,Z 354.46,A -85,B 0,C 180,E1 -3890.651,E2 -3890.651} C_VEL
LIN {X 0,Y 538.028,Z 354.462,A -85,B 0,C 180,E1 -3893.887,E2 -3893.887} C_VEL
LIN {X 0,Y 538.045,Z 354.458,A -85,B 0,C 180,E1 -3896.366,E2 -3896.366} C_VEL
LIN {X 0,Y 538.034,Z 354.465,A -85,B 0,C 180,E1 -3898.933,E2 -3898.933} C_VEL
LIN {X 0,Y 538.029,Z 354.461,A -85,B 0,C 180,E1 -3901.889,E2 -3901.889} C_VEL
LIN {X 0,Y 538.033,Z 354.462,A -85,B 0,C 180,E1 -3904.62,E2 -3904.62} C_VEL
LIN {X 0,Y 538.009,Z 354.472,A -85,B 0,C 180,E1 -3907.17,E2 -3907.17} C_VEL
LIN {X 0,Y 538.03,Z 354.461,A -85,B 0,C 180,E1 -3909.795,E2 -3909.795} C_VEL
LIN {X 0,Y 538.018,Z 354.467,A -85,B 0,C 180,E1 -3912.785,E2 -3912.785} C_VEL
LIN {X 0,Y 538.031,Z 354.468,A -85,B 0,C 180,E1 -3915.14,E2 -3915.14} C_VEL
LIN {X 0,Y 538.038,Z 354.46,A -85,B 0,C 180,E1 -3918.227,E2 -3918.227} C_VEL
LIN {X 0,Y 538.012,Z 354.469,A -85,B 0,C 180,E1 -3921.169,E2 -3921.169} C_VEL
LIN {X 0,Y 538.025,Z 354.461,A -85,B 0,C 180,E1 -3924.082,E2 -3924.082} C_VEL
LIN {X 0,Y 538.026,Z 354.467,A -85,B 0,C 180,E1 -3926.727,E2 -3926.727} C_VEL
LIN {X 0,Y 538.02,Z 354.462,A -85,B 0,C 180,E1 -3929.555,E2 -3929.555} C_VEL
LIN {X 0,Y 538.042,Z 354.459,A -85,B 0,C 180,E1 -3931.95,E2 -3931.95} C_VEL
LIN {X 0,Y 538.069,Z 354.46,A -85,B 0,C 180,E1 -3934.467,E2 -3934.467} C_VEL
LIN {X 0,Y 538.017,Z 354.469,A -85,B 0,C 180,E1 -3936.928,E2 -3936.928} C_VEL
LIN {X 0,Y 538.071,Z 354.457,A -85,B 0,C 180,E1 -3940.147,E2 -3940.147} C_VEL
LIN {X 0,Y 538.02,Z 354.463,A -85,B 0,C 180,E1 -3943.299,E2 -3943.299} C_VEL
LIN {X 0,Y 538.056,Z 354.457,A -85,B 0,C 180,E1 -3945.63,E2 -3945.63} C_VEL
LIN {X 0,Y 538.081,Z 354.463,A -85,B 0,C 180,E1 -3948.701,E2 -3948.701} C_VEL
LIN {X 0,Y 538.082,Z 354.454,A -85,B 0,C 180,E1 -3951.739,E2 -3951.739} C_VEL
LIN {X 0,Y 538.176,Z 354.449,A -85,B 0,C 180,E1 -3954.755,E2 -3954.755} C_VEL
LIN {X 0,Y 538.159,Z 354.444,A -85,B 0,C 180,E1 -3957.754,E2 -3957.754} C_VEL
LIN {X 0,Y 538.177,Z 354.448,A -85,B 0,C 180,E1 -3960.748,E2 -3960.748} C_VEL
LIN {X 0,Y 538.134,Z 354.45,A -85,B 0,C 180,E1 -3962.994,E2 -3962.994} C_VEL
LIN {X 0,Y 538.115,Z 354.452,A -85,B 0,C 180,E1 -3965.997,E2 -3965.997} C_VEL
LIN {X 0,Y 538.068,Z 354.457,A -85,B 0,C 180,E1 -3969.018,E2 -3969.018} C_VEL
LIN {X 0,Y 538.074,Z 354.459,A -85,B 0,C 180,E1 -3972.063,E2 -3972.063} C_VEL
LIN {X 0,Y 538.037,Z 354.46,A -85,B 0,C 180,E1 -3975.144,E2 -3975.144} C_VEL
LIN {X 0,Y 538.027,Z 354.47,A -85,B 0,C 180,E1 -3978.27,E2 -3978.27} C_VEL
LIN {X 0,Y 538.034,Z 354.464,A -85,B 0,C 180,E1 -3980.652,E2 -3980.652} C_VEL
LIN {X 0,Y 538.015,Z 354.466,A -85,B 0,C 180,E1 -3983.888,E2 -3983.888} C_VEL
LIN {X 0,Y 538.042,Z 354.466,A -85,B 0,C 180,E1 -3986.367,E2 -3986.367} C_VEL
LIN {X 0,Y 538.049,Z 354.458,A -85,B 0,C 180,E1 -3988.939,E2 -3988.939} C_VEL
LIN {X 0,Y 538.021,Z 354.466,A -85,B 0,C 180,E1 -3991.891,E2 -3991.891} C_VEL
LIN {X 0,Y 538.027,Z 354.463,A -85,B 0,C 180,E1 -3994.622,E2 -3994.622} C_VEL
LIN {X 0,Y 538.002,Z 354.464,A -85,B 0,C 180,E1 -3997.171,E2 -3997.171} C_VEL
LIN {X 0,Y 538.049,Z 354.463,A -85,B 0,C 180,E1 -3999.795,E2 -3999.795} C_VEL
LIN {X 0,Y 538.019,Z 354.462,A -85,B 0,C 180,E1 -4002.786,E2 -4002.786} C_VEL
LIN {X 0,Y 538.026,Z 354.469,A -85,B 0,C 180,E1 -4005.926,E2 -4005.926} C_VEL
LIN {X 0,Y 538.075,Z 354.455,A -85,B 0,C 180,E1 -4009.25,E2 -4009.25} C_VEL
LIN {X 0,Y 537.992,Z 354.471,A -85,B 0,C 180,E1 -4012.123,E2 -4012.123} C_VEL
LIN {X 0,Y 538.019,Z 354.461,A -85,B 0,C 180,E1 -4014.918,E2 -4014.918} C_VEL
LIN {X 0,Y 538.031,Z 354.465,A -85,B 0,C 180,E1 -4017.619,E2 -4017.619} C_VEL
LIN {X 0,Y 538.043,Z 354.465,A -85,B 0,C 180,E1 -4020.241,E2 -4020.241} C_VEL
LIN {X 0,Y 538.067,Z 354.459,A -85,B 0,C 180,E1 -4022.797,E2 -4022.797} C_VEL
LIN {X 0,Y 538.075,Z 354.578,A -85,B 0,C 180,E1 -4025.269,E2 -4025.269} C_VEL
LIN {X 0,Y 539.504,Z 362.887,A -85,B 0,C 180,E1 -4026.59,E2 -4026.59} C_VEL
LIN {X 0,Y 539.033,Z 381.766,A -85,B 0,C 180,E1 -4029.389,E2 -4029.389} C_VEL
LIN {X 0,Y 538.705,Z 401.365,A -85,B 0,C 180,E1 -4032.245,E2 -4032.245} C_VEL
LIN {X 0,Y 538.426,Z 422.422,A -85,B 0,C 180,E1 -4035.251,E2 -4035.251} C_VEL
LIN {X 0,Y 539.704,Z 431.874,A -85,B 0,C 180,E1 -4035.413,E2 -4035.413} C_VEL
LIN {X 0,Y 539.346,Z 530.701,A -85,B 0,C 180,E1 -4036.747,E2 -4036.747} C_VEL
LIN {X 0,Y 539.144,Z 543.24,A -85,B 0,C 180,E1 -4037.053,E2 -4037.053} C_VEL
LIN {X 0,Y 538.939,Z 556.196,A -85,B 0,C 180,E1 -4037.527,E2 -4037.527} C_VEL
LIN {X 0,Y 538.719,Z 568.089,A -85,B 0,C 180,E1 -4038.119,E2 -4038.119} C_VEL
LIN {X 0,Y 538.511,Z 580.133,A -85,B 0,C 180,E1 -4038.902,E2 -4038.902} C_VEL
LIN {X 0,Y 538.262,Z 590.602,A -85,B 0,C 180,E1 -4039.753,E2 -4039.753} C_VEL
LIN {X 0,Y 538.067,Z 599.115,A -85,B 0,C 180,E1 -4040.603,E2 -4040.603} C_VEL
LIN {X 0,Y 537.921,Z 606.962,A -85,B 0,C 180,E1 -4041.548,E2 -4041.548} C_VEL
LIN {X 0,Y 537.754,Z 614.622,A -85,B 0,C 180,E1 -4042.679,E2 -4042.679} C_VEL
LIN {X 0,Y 537.693,Z 621.68,A -85,B 0,C 180,E1 -4043.998,E2 -4043.998} C_VEL
LIN {X 0,Y 537.54,Z 626.373,A -85,B 0,C 180,E1 -4045.125,E2 -4045.125} C_VEL
LIN {X 0,Y 537.591,Z 629.958,A -85,B 0,C 180,E1 -4046.252,E2 -4046.252} C_VEL
LIN {X 0,Y 537.551,Z 631.807,A -85,B 0,C 180,E1 -4047.002,E2 -4047.002} C_VEL
LIN {X 0,Y 537.451,Z 634.182,A -85,B 0,C 180,E1 -4048.501,E2 -4048.501} C_VEL
LIN {X 0,Y 537.442,Z 635,A -85,B 0,C 180,E1 -4050,E2 -4050} C_VEL
LIN {X 0,Y 537.451,Z 634.184,A -85,B 0,C 180,E1 -4051.499,E2 -4051.499} C_VEL
LIN {X 0,Y 537.551,Z 631.81,A -85,B 0,C 180,E1 -4052.998,E2 -4052.998} C_VEL
LIN {X 0,Y 537.603,Z 628.895,A -85,B 0,C 180,E1 -4054.123,E2 -4054.123} C_VEL
LIN {X 0,Y 537.588,Z 624.948,A -85,B 0,C 180,E1 -4055.251,E2 -4055.251} C_VEL
LIN {X 0,Y 537.644,Z 620.125,A -85,B 0,C 180,E1 -4056.326,E2 -4056.326} C_VEL
LIN {X 0,Y 537.79,Z 613.467,A -85,B 0,C 180,E1 -4057.509,E2 -4057.509} C_VEL
LIN {X 0,Y 537.972,Z 605.478,A -85,B 0,C 180,E1 -4058.64,E2 -4058.64} C_VEL
LIN {X 0,Y 538.143,Z 597.335,A -85,B 0,C 180,E1 -4059.585,E2 -4059.585} C_VEL
LIN {X 0,Y 538.383,Z 587.381,A -85,B 0,C 180,E1 -4060.53,E2 -4060.53} C_VEL
LIN {X 0,Y 538.565,Z 577.516,A -85,B 0,C 180,E1 -4061.288,E2 -4061.288} C_VEL
LIN {X 0,Y 538.731,Z 566.407,A -85,B 0,C 180,E1 -4061.973,E2 -4061.973} C_VEL
LIN {X 0,Y 538.966,Z 553.912,A -85,B 0,C 180,E1 -4062.568,E2 -4062.568} C_VEL
LIN {X 0,Y 539.202,Z 540.852,A -85,B 0,C 180,E1 -4063.017,E2 -4063.017} C_VEL
LIN {X 0,Y 539.387,Z 527.834,A -85,B 0,C 180,E1 -4063.3,E2 -4063.3} C_VEL
LIN {X 0,Y 539.548,Z 429.861,A -85,B 0,C 180,E1 -4064.618,E2 -4064.618} C_VEL
LIN {X 0,Y 538.386,Z 422.157,A -85,B 0,C 180,E1 -4064.754,E2 -4064.754} C_VEL
LIN {X 0,Y 538.753,Z 398.993,A -85,B 0,C 180,E1 -4068.09,E2 -4068.09} C_VEL
LIN {X 0,Y 539.158,Z 377.612,A -85,B 0,C 180,E1 -4071.206,E2 -4071.206} C_VEL
LIN {X 0,Y 539.402,Z 361.425,A -85,B 0,C 180,E1 -4073.618,E2 -4073.618} C_VEL
LIN {X 0,Y 538.08,Z 354.461,A -85,B 0,C 180,E1 -4074.757,E2 -4074.757} C_VEL
LIN {X 0,Y 538.061,Z 354.46,A -85,B 0,C 180,E1 -4077.352,E2 -4077.352} C_VEL
LIN {X 0,Y 538.043,Z 354.465,A -85,B 0,C 180,E1 -4079.759,E2 -4079.759} C_VEL
LIN {X 0,Y 538.031,Z 354.466,A -85,B 0,C 180,E1 -4082.381,E2 -4082.381} C_VEL
LIN {X 0,Y 538.019,Z 354.462,A -85,B 0,C 180,E1 -4085.082,E2 -4085.082} C_VEL
LIN {X 0,Y 537.992,Z 354.474,A -85,B 0,C 180,E1 -4087.877,E2 -4087.877} C_VEL
LIN {X 0,Y 538.075,Z 354.456,A -85,B 0,C 180,E1 -4090.772,E2 -4090.772} C_VEL
LIN {X 0,Y 538.026,Z 354.469,A -85,B 0,C 180,E1 -4094.074,E2 -4094.074} C_VEL
LIN {X 0,Y 538.019,Z 354.463,A -85,B 0,C 180,E1 -4097.214,E2 -4097.214} C_VEL
LIN {X 0,Y 538.049,Z 354.462,A -85,B 0,C 180,E1 -4100.205,E2 -4100.205} C_VEL
LIN {X 0,Y 538.023,Z 354.461,A -85,B 0,C 180,E1 -4103.067,E2 -4103.067} C_VEL
LIN {X 0,Y 538.026,Z 354.468,A -85,B 0,C 180,E1 -4105.827,E2 -4105.827} C_VEL
LIN {X 0,Y 538.017,Z 354.463,A -85,B 0,C 180,E1 -4108.499,E2 -4108.499} C_VEL
LIN {X 0,Y 538.051,Z 354.458,A -85,B 0,C 180,E1 -4111.099,E2 -4111.099} C_VEL
LIN {X 0,Y 538.042,Z 354.466,A -85,B 0,C 180,E1 -4113.633,E2 -4113.633} C_VEL
LIN {X 0,Y 538.014,Z 354.465,A -85,B 0,C 180,E1 -4116.118,E2 -4116.118} C_VEL
LIN {X 0,Y 538.034,Z 354.464,A -85,B 0,C 180,E1 -4119.348,E2 -4119.348} C_VEL
LIN {X 0,Y 538.063,Z 354.454,A -85,B 0,C 180,E1 -4122.517,E2 -4122.517} C_VEL
LIN {X 0,Y 538.054,Z 354.465,A -85,B 0,C 180,E1 -4125.631,E2 -4125.631} C_VEL
LIN {X 0,Y 538.08,Z 354.454,A -85,B 0,C 180,E1 -4128.702,E2 -4128.702} C_VEL
LIN {X 0,Y 538.082,Z 354.456,A -85,B 0,C 180,E1 -4131.74,E2 -4131.74} C_VEL
LIN {X 0,Y 538.158,Z 354.446,A -85,B 0,C 180,E1 -4134.755,E2 -4134.755} C_VEL
LIN {X 0,Y 538.159,Z 354.447,A -85,B 0,C 180,E1 -4137.755,E2 -4137.755} C_VEL
LIN {X 0,Y 538.178,Z 354.444,A -85,B 0,C 180,E1 -4140.748,E2 -4140.748} C_VEL
LIN {X 0,Y 538.137,Z 354.45,A -85,B 0,C 180,E1 -4142.995,E2 -4142.995} C_VEL
LIN {X 0,Y 538.117,Z 354.45,A -85,B 0,C 180,E1 -4145.998,E2 -4145.998} C_VEL
LIN {X 0,Y 538.07,Z 354.461,A -85,B 0,C 180,E1 -4149.018,E2 -4149.018} C_VEL
LIN {X 0,Y 538.076,Z 354.453,A -85,B 0,C 180,E1 -4152.063,E2 -4152.063} C_VEL
LIN {X 0,Y 538.038,Z 354.467,A -85,B 0,C 180,E1 -4155.144,E2 -4155.144} C_VEL
LIN {X 0,Y 538.03,Z 354.461,A -85,B 0,C 180,E1 -4158.271,E2 -4158.271} C_VEL
LIN {X 0,Y 538.036,Z 354.462,A -85,B 0,C 180,E1 -4160.652,E2 -4160.652} C_VEL
LIN {X 0,Y 538.034,Z 354.458,A -85,B 0,C 180,E1 -4163.887,E2 -4163.887} C_VEL
LIN {X 0,Y 538.044,Z 354.46,A -85,B 0,C 180,E1 -4166.367,E2 -4166.367} C_VEL
LIN {X 0,Y 538.027,Z 354.47,A -85,B 0,C 180,E1 -4168.935,E2 -4168.935} C_VEL
LIN {X 0,Y 538.023,Z 354.462,A -85,B 0,C 180,E1 -4171.891,E2 -4171.891} C_VEL
LIN {X 0,Y 538.03,Z 354.463,A -85,B 0,C 180,E1 -4174.622,E2 -4174.622} C_VEL
LIN {X 0,Y 538.004,Z 354.468,A -85,B 0,C 180,E1 -4177.172,E2 -4177.172} C_VEL
LIN {X 0,Y 538.032,Z 354.463,A -85,B 0,C 180,E1 -4180.278,E2 -4180.278} C_VEL
LIN {X 0,Y 537.393,Z 354.548,A -85,B 0,C 180,E1 -4180.904,E2 -4180.904} C_VEL
LIN {X 0,Y 534.539,Z 354.904,A -85,B 0,C 180,E1 -4181.918,E2 -4181.918} C_VEL
LIN {X 0,Y 532.104,Z 355.205,A -85,B 0,C 180,E1 -4182.735,E2 -4182.735} C_VEL
LIN {X 0,Y 531.05,Z 355.333,A -85,B 0,C 180,E1 -4183.366,E2 -4183.366} C_VEL
LIN {X 0,Y 530.962,Z 355.343,A -85,B 0,C 180,E1 -4183.58,E2 -4183.58} C_VEL
LIN {X 0,Y 530.965,Z 355.348,A -85,B 0,C 180,E1 -4186.507,E2 -4186.507} C_VEL
LIN {X 0,Y 530.989,Z 355.344,A -85,B 0,C 180,E1 -4188.977,E2 -4188.977} C_VEL
LIN {X 0,Y 530.96,Z 355.345,A -85,B 0,C 180,E1 -4191.531,E2 -4191.531} C_VEL
LIN {X 0,Y 530.991,Z 355.348,A -85,B 0,C 180,E1 -4194.384,E2 -4194.384} C_VEL
LIN {X 0,Y 531.043,Z 355.485,A -85,B 0,C 180,E1 -4194.997,E2 -4194.997} C_VEL
LIN {X 0,Y 531.542,Z 360.447,A -85,B 0,C 180,E1 -4196.04,E2 -4196.04} C_VEL
LIN {X 0,Y 531.222,Z 375.733,A -85,B 0,C 180,E1 -4199.118,E2 -4199.118} C_VEL
LIN {X 0,Y 532.805,Z 384.25,A -85,B 0,C 180,E1 -4199.281,E2 -4199.281} C_VEL
LIN {X 0,Y 532.438,Z 482.045,A -85,B 0,C 180,E1 -4200.626,E2 -4200.626} C_VEL
LIN {X 0,Y 532.212,Z 495.446,A -85,B 0,C 180,E1 -4200.969,E2 -4200.969} C_VEL
LIN {X 0,Y 532.029,Z 507.866,A -85,B 0,C 180,E1 -4201.444,E2 -4201.444} C_VEL
LIN {X 0,Y 531.785,Z 518.865,A -85,B 0,C 180,E1 -4202.008,E2 -4202.008} C_VEL
LIN {X 0,Y 531.559,Z 530.195,A -85,B 0,C 180,E1 -4202.756,E2 -4202.756} C_VEL
LIN {X 0,Y 531.297,Z 540.348,A -85,B 0,C 180,E1 -4203.591,E2 -4203.591} C_VEL
LIN {X 0,Y 531.073,Z 549.628,A -85,B 0,C 180,E1 -4204.527,E2 -4204.527} C_VEL
LIN {X 0,Y 530.877,Z 557.989,A -85,B 0,C 180,E1 -4205.563,E2 -4205.563} C_VEL
LIN {X 0,Y 530.684,Z 565.984,A -85,B 0,C 180,E1 -4206.798,E2 -4206.798} C_VEL
LIN {X 0,Y 530.583,Z 572.188,A -85,B 0,C 180,E1 -4208.005,E2 -4208.005} C_VEL
LIN {X 0,Y 530.498,Z 576.405,A -85,B 0,C 180,E1 -4209.042,E2 -4209.042} C_VEL
LIN {X 0,Y 530.468,Z 579.961,A -85,B 0,C 180,E1 -4210.164,E2 -4210.164} C_VEL
LIN {X 0,Y 530.372,Z 582.882,A -85,B 0,C 180,E1 -4211.457,E2 -4211.457} C_VEL
LIN {X 0,Y 530.385,Z 584.414,A -85,B 0,C 180,E1 -4212.566,E2 -4212.566} C_VEL
LIN {X 0,Y 530.331,Z 585.147,A -85,B 0,C 180,E1 -4213.842,E2 -4213.842} C_VEL
LIN {X 0,Y 530.395,Z 584.637,A -85,B 0,C 180,E1 -4215.306,E2 -4215.306} C_VEL
LIN {X 0,Y 530.396,Z 583.568,A -85,B 0,C 180,E1 -4216.202,E2 -4216.202} C_VEL
LIN {X 0,Y 530.387,Z 582.216,A -85,B 0,C 180,E1 -4216.982,E2 -4216.982} C_VEL
LIN {X 0,Y 530.472,Z 579.336,A -85,B 0,C 180,E1 -4218.15,E2 -4218.15} C_VEL
LIN {X 0,Y 530.504,Z 575.425,A -85,B 0,C 180,E1 -4219.312,E2 -4219.312} C_VEL
LIN {X 0,Y 530.604,Z 570.372,A -85,B 0,C 180,E1 -4220.47,E2 -4220.47} C_VEL
LIN {X 0,Y 530.74,Z 564.02,A -85,B 0,C 180,E1 -4221.625,E2 -4221.625} C_VEL
LIN {X 0,Y 530.936,Z 556.087,A -85,B 0,C 180,E1 -4222.776,E2 -4222.776} C_VEL
LIN {X 0,Y 531.105,Z 547.844,A -85,B 0,C 180,E1 -4223.754,E2 -4223.754} C_VEL
LIN {X 0,Y 531.325,Z 538.247,A -85,B 0,C 180,E1 -4224.687,E2 -4224.687} C_VEL
LIN {X 0,Y 531.595,Z 527.245,A -85,B 0,C 180,E1 -4225.545,E2 -4225.545} C_VEL
LIN {X 0,Y 531.856,Z 516.486,A -85,B 0,C 180,E1 -4226.212,E2 -4226.212} C_VEL
LIN {X 0,Y 532.083,Z 504.655,A -85,B 0,C 180,E1 -4226.782,E2 -4226.782} C_VEL
LIN {X 0,Y 532.291,Z 491.768,A -85,B 0,C 180,E1 -4227.233,E2 -4227.233} C_VEL
LIN {X 0,Y 532.443,Z 478.954,A -85,B 0,C 180,E1 -4227.518,E2 -4227.518} C_VEL
LIN {X 0,Y 532.742,Z 383.614,A -85,B 0,C 180,E1 -4228.819,E2 -4228.819} C_VEL
LIN {X 0,Y 531.134,Z 375.481,A -85,B 0,C 180,E1 -4228.981,E2 -4228.981} C_VEL
LIN {X 0,Y 531.442,Z 363.007,A -85,B 0,C 180,E1 -4231.516,E2 -4231.516} C_VEL
LIN {X 0,Y 531.429,Z 357.442,A -85,B 0,C 180,E1 -4232.653,E2 -4232.653} C_VEL
LIN {X 0,Y 531.069,Z 355.337,A -85,B 0,C 180,E1 -4233.129,E2 -4233.129} C_VEL
LIN {X 0,Y 531.075,Z 355.33,A -85,B 0,C 180,E1 -4236.077,E2 -4236.077} C_VEL
LIN {X 0,Y 531.029,Z 355.339,A -85,B 0,C 180,E1 -4239.138,E2 -4239.138} C_VEL
LIN {X 0,Y 531.047,Z 355.33,A -85,B 0,C 180,E1 -4242.225,E2 -4242.225} C_VEL
LIN {X 0,Y 531,Z 355.346,A -85,B 0,C 180,E1 -4245.349,E2 -4245.349} C_VEL
LIN {X 0,Y 530.993,Z 355.337,A -85,B 0,C 180,E1 -4248.521,E2 -4248.521} C_VEL
LIN {X 0,Y 531.003,Z 355.34,A -85,B 0,C 180,E1 -4250.937,E2 -4250.937} C_VEL
LIN {X 0,Y 530.984,Z 355.338,A -85,B 0,C 180,E1 -4254.224,E2 -4254.224} C_VEL
LIN {X 0,Y 531.005,Z 355.338,A -85,B 0,C 180,E1 -4256.743,E2 -4256.743} C_VEL
LIN {X 0,Y 530.985,Z 355.345,A -85,B 0,C 180,E1 -4259.322,E2 -4259.322} C_VEL
LIN {X 0,Y 530.982,Z 355.338,A -85,B 0,C 180,E1 -4262.102,E2 -4262.102} C_VEL
LIN {X 0,Y 530.991,Z 355.342,A -85,B 0,C 180,E1 -4264.853,E2 -4264.853} C_VEL
LIN {X 0,Y 530.967,Z 355.344,A -85,B 0,C 180,E1 -4267.507,E2 -4267.507} C_VEL
LIN {X 0,Y 530.984,Z 355.339,A -85,B 0,C 180,E1 -4270.431,E2 -4270.431} C_VEL
LIN {X 0,Y 530.965,Z 355.346,A -85,B 0,C 180,E1 -4273.281,E2 -4273.281} C_VEL
LIN {X 0,Y 530.986,Z 355.339,A -85,B 0,C 180,E1 -4275.62,E2 -4275.62} C_VEL
LIN {X 0,Y 530.998,Z 355.339,A -85,B 0,C 180,E1 -4278.564,E2 -4278.564} C_VEL
LIN {X 0,Y 530.956,Z 355.343,A -85,B 0,C 180,E1 -4281.529,E2 -4281.529} C_VEL
LIN {X 0,Y 530.977,Z 355.341,A -85,B 0,C 180,E1 -4284.381,E2 -4284.381} C_VEL
LIN {X 0,Y 530.967,Z 355.346,A -85,B 0,C 180,E1 -4287.133,E2 -4287.133} C_VEL
LIN {X 0,Y 530.964,Z 355.34,A -85,B 0,C 180,E1 -4289.802,E2 -4289.802} C_VEL
LIN {X 0,Y 531.012,Z 355.338,A -85,B 0,C 180,E1 -4292.465,E2 -4292.465} C_VEL
LIN {X 0,Y 531.001,Z 355.343,A -85,B 0,C 180,E1 -4294.942,E2 -4294.942} C_VEL
LIN {X 0,Y 530.964,Z 355.343,A -85,B 0,C 180,E1 -4298.246,E2 -4298.246} C_VEL
LIN {X 0,Y 530.99,Z 355.346,A -85,B 0,C 180,E1 -4300.677,E2 -4300.677} C_VEL
LIN {X 0,Y 530.985,Z 355.342,A -85,B 0,C 180,E1 -4303.071,E2 -4303.071} C_VEL
LIN {X 0,Y 531.01,Z 355.335,A -85,B 0,C 180,E1 -4305.435,E2 -4305.435} C_VEL
LIN {X 0,Y 531.038,Z 355.339,A -85,B 0,C 180,E1 -4308.549,E2 -4308.549} C_VEL
LIN {X 0,Y 531.051,Z 355.329,A -85,B 0,C 180,E1 -4311.629,E2 -4311.629} C_VEL
LIN {X 0,Y 531.132,Z 355.327,A -85,B 0,C 180,E1 -4314.685,E2 -4314.685} C_VEL
LIN {X 0,Y 531.131,Z 355.32,A -85,B 0,C 180,E1 -4317.725,E2 -4317.725} C_VEL
LIN {X 0,Y 531.147,Z 355.323,A -85,B 0,C 180,E1 -4320.758,E2 -4320.758} C_VEL
LIN {X 0,Y 531.101,Z 355.325,A -85,B 0,C 180,E1 -4323.034,E2 -4323.034} C_VEL
LIN {X 0,Y 531.075,Z 355.33,A -85,B 0,C 180,E1 -4326.077,E2 -4326.077} C_VEL
LIN {X 0,Y 531.027,Z 355.333,A -85,B 0,C 180,E1 -4329.138,E2 -4329.138} C_VEL
LIN {X 0,Y 531.032,Z 355.339,A -85,B 0,C 180,E1 -4332.225,E2 -4332.225} C_VEL
LIN {X 0,Y 530.987,Z 355.337,A -85,B 0,C 180,E1 -4335.35,E2 -4335.35} C_VEL
LIN {X 0,Y 531.007,Z 355.336,A -85,B 0,C 180,E1 -4337.723,E2 -4337.723} C_VEL
LIN {X 0,Y 530.993,Z 355.338,A -85,B 0,C 180,E1 -4340.938,E2 -4340.938} C_VEL
LIN {X 0,Y 530.972,Z 355.349,A -85,B 0,C 180,E1 -4344.225,E2 -4344.225} C_VEL
LIN {X 0,Y 531.004,Z 355.338,A -85,B 0,C 180,E1 -4346.744,E2 -4346.744} C_VEL
LIN {X 0,Y 530.993,Z 355.337,A -85,B 0,C 180,E1 -4349.322,E2 -4349.322} C_VEL
LIN {X 0,Y 530.974,Z 355.348,A -85,B 0,C 180,E1 -4352.104,E2 -4352.104} C_VEL
LIN {X 0,Y 530.984,Z 355.339,A -85,B 0,C 180,E1 -4354.855,E2 -4354.855} C_VEL
LIN {X 0,Y 530.961,Z 355.342,A -85,B 0,C 180,E1 -4357.508,E2 -4357.508} C_VEL
LIN {X 0,Y 531.021,Z 355.337,A -85,B 0,C 180,E1 -4360.429,E2 -4360.429} C_VEL
LIN {X 0,Y 530.961,Z 355.343,A -85,B 0,C 180,E1 -4363.495,E2 -4363.495} C_VEL
LIN {X 0,Y 530.961,Z 355.343,A -85,B 0,C 180,E1 -4366.506,E2 -4366.506} C_VEL
LIN {X 0,Y 531.024,Z 355.336,A -85,B 0,C 180,E1 -4369.572,E2 -4369.572} C_VEL
LIN {X 0,Y 530.967,Z 355.341,A -85,B 0,C 180,E1 -4372.577,E2 -4372.577} C_VEL
LIN {X 0,Y 531.001,Z 355.337,A -85,B 0,C 180,E1 -4375.312,E2 -4375.312} C_VEL
LIN {X 0,Y 530.982,Z 355.345,A -85,B 0,C 180,E1 -4378.034,E2 -4378.034} C_VEL
LIN {X 0,Y 531.007,Z 355.338,A -85,B 0,C 180,E1 -4380.871,E2 -4380.871} C_VEL
LIN {X 0,Y 531.007,Z 355.341,A -85,B 0,C 180,E1 -4383.257,E2 -4383.257} C_VEL
LIN {X 0,Y 531.052,Z 355.491,A -85,B 0,C 180,E1 -4385.102,E2 -4385.102} C_VEL
LIN {X 0,Y 532.577,Z 363.973,A -85,B 0,C 180,E1 -4386.473,E2 -4386.473} C_VEL
LIN {X 0,Y 532.062,Z 382.796,A -85,B 0,C 180,E1 -4389.302,E2 -4389.302} C_VEL
LIN {X 0,Y 531.704,Z 401.834,A -85,B 0,C 180,E1 -4392.118,E2 -4392.118} C_VEL
LIN {X 0,Y 531.375,Z 421.829,A -85,B 0,C 180,E1 -4395.043,E2 -4395.043} C_VEL
LIN {X 0,Y 532.821,Z 432.375,A -85,B 0,C 180,E1 -4395.232,E2 -4395.232} C_VEL
LIN {X 0,Y 532.43,Z 530.328,A -85,B 0,C 180,E1 -4396.572,E2 -4396.572} C_VEL
LIN {X 0,Y 532.191,Z 543.645,A -85,B 0,C 180,E1 -4396.906,E2 -4396.906} C_VEL
LIN {X 0,Y 531.983,Z 555.844,A -85,B 0,C 180,E1 -4397.361,E2 -4397.361} C_VEL
LIN {X 0,Y 531.725,Z 568.127,A -85,B 0,C 180,E1 -4397.983,E2 -4397.983} C_VEL
LIN {X 0,Y 531.502,Z 579.79,A -85,B 0,C 180,E1 -4398.753,E2 -4398.753} C_VEL
LIN {X 0,Y 531.22,Z 590.265,A -85,B 0,C 180,E1 -4399.615,E2 -4399.615} C_VEL
LIN {X 0,Y 531.033,Z 598.833,A -85,B 0,C 180,E1 -4400.478,E2 -4400.478} C_VEL
LIN {X 0,Y 530.886,Z 606.742,A -85,B 0,C 180,E1 -4401.435,E2 -4401.435} C_VEL
LIN {X 0,Y 530.681,Z 614.465,A -85,B 0,C 180,E1 -4402.581,E2 -4402.581} C_VEL
LIN {X 0,Y 530.604,Z 621.589,A -85,B 0,C 180,E1 -4403.918,E2 -4403.918} C_VEL
LIN {X 0,Y 530.459,Z 626.325,A -85,B 0,C 180,E1 -4405.06,E2 -4405.06} C_VEL
LIN {X 0,Y 530.516,Z 629.947,A -85,B 0,C 180,E1 -4406.202,E2 -4406.202} C_VEL
LIN {X 0,Y 530.457,Z 631.804,A -85,B 0,C 180,E1 -4406.962,E2 -4406.962} C_VEL
LIN {X 0,Y 530.41,Z 633.192,A -85,B 0,C 180,E1 -4407.722,E2 -4407.722} C_VEL
LIN {X 0,Y 530.344,Z 634.785,A -85,B 0,C 180,E1 -4409.241,E2 -4409.241} C_VEL
LIN {X 0,Y 530.342,Z 635,A -85,B 0,C 180,E1 -4410,E2 -4410} C_VEL
LIN {X 0,Y 530.361,Z 634.183,A -85,B 0,C 180,E1 -4411.519,E2 -4411.519} C_VEL
LIN {X 0,Y 530.41,Z 633.195,A -85,B 0,C 180,E1 -4412.278,E2 -4412.278} C_VEL
LIN {X 0,Y 530.457,Z 631.807,A -85,B 0,C 180,E1 -4413.038,E2 -4413.038} C_VEL
LIN {X 0,Y 530.522,Z 628.876,A -85,B 0,C 180,E1 -4414.178,E2 -4414.178} C_VEL
LIN {X 0,Y 530.525,Z 624.887,A -85,B 0,C 180,E1 -4415.321,E2 -4415.321} C_VEL
LIN {X 0,Y 530.595,Z 619.161,A -85,B 0,C 180,E1 -4416.579,E2 -4416.579} C_VEL
LIN {X 0,Y 530.733,Z 612.054,A -85,B 0,C 180,E1 -4417.801,E2 -4417.801} C_VEL
LIN {X 0,Y 530.93,Z 603.743,A -85,B 0,C 180,E1 -4418.948,E2 -4418.948} C_VEL
LIN {X 0,Y 531.122,Z 595.224,A -85,B 0,C 180,E1 -4419.905,E2 -4419.905} C_VEL
LIN {X 0,Y 531.38,Z 584.703,A -85,B 0,C 180,E1 -4420.863,E2 -4420.863} C_VEL
LIN {X 0,Y 531.66,Z 572.732,A -85,B 0,C 180,E1 -4421.735,E2 -4421.735} C_VEL
LIN {X 0,Y 531.927,Z 560.963,A -85,B 0,C 180,E1 -4422.398,E2 -4422.398} C_VEL
LIN {X 0,Y 532.135,Z 548.585,A -85,B 0,C 180,E1 -4422.926,E2 -4422.926} C_VEL
LIN {X 0,Y 532.339,Z 535.887,A -85,B 0,C 180,E1 -4423.309,E2 -4423.309} C_VEL
LIN {X 0,Y 532.465,Z 520.826,A -85,B 0,C 180,E1 -4423.573,E2 -4423.573} C_VEL
LIN {X 0,Y 532.717,Z 430.842,A -85,B 0,C 180,E1 -4424.792,E2 -4424.792} C_VEL
LIN {X 0,Y 531.339,Z 421.718,A -85,B 0,C 180,E1 -4424.966,E2 -4424.966} C_VEL
LIN {X 0,Y 531.743,Z 400.096,A -85,B 0,C 180,E1 -4428.125,E2 -4428.125} C_VEL
LIN {X 0,Y 532.137,Z 380.027,A -85,B 0,C 180,E1 -4431.093,E2 -4431.093} C_VEL
LIN {X 0,Y 532.517,Z 363.837,A -85,B 0,C 180,E1 -4433.529,E2 -4433.529} C_VEL
LIN {X 0,Y 531.053,Z 355.335,A -85,B 0,C 180,E1 -4434.924,E2 -4434.924} C_VEL
LIN {X 0,Y 531.017,Z 355.339,A -85,B 0,C 180,E1 -4437.595,E2 -4437.595} C_VEL
LIN {X 0,Y 530.982,Z 355.342,A -85,B 0,C 180,E1 -4440.646,E2 -4440.646} C_VEL
LIN {X 0,Y 530.99,Z 355.342,A -85,B 0,C 180,E1 -4443.772,E2 -4443.772} C_VEL
LIN {X 0,Y 530.967,Z 355.344,A -85,B 0,C 180,E1 -4446.557,E2 -4446.557} C_VEL
LIN {X 0,Y 531.022,Z 355.34,A -85,B 0,C 180,E1 -4449.859,E2 -4449.859} C_VEL
LIN {X 0,Y 530.977,Z 355.341,A -85,B 0,C 180,E1 -4452.456,E2 -4452.456} C_VEL
LIN {X 0,Y 530.983,Z 355.343,A -85,B 0,C 180,E1 -4455.62,E2 -4455.62} C_VEL
LIN {X 0,Y 531.002,Z 355.337,A -85,B 0,C 180,E1 -4458.565,E2 -4458.565} C_VEL
LIN {X 0,Y 530.963,Z 355.343,A -85,B 0,C 180,E1 -4461.345,E2 -4461.345} C_VEL
LIN {X 0,Y 530.976,Z 355.341,A -85,B 0,C 180,E1 -4464.382,E2 -4464.382} C_VEL
LIN {X 0,Y 530.968,Z 355.34,A -85,B 0,C 180,E1 -4467.133,E2 -4467.133} C_VEL
LIN {X 0,Y 530.979,Z 355.345,A -85,B 0,C 180,E1 -4469.804,E2 -4469.804} C_VEL
LIN {X 0,Y 531.01,Z 355.335,A -85,B 0,C 180,E1 -4472.466,E2 -4472.466} C_VEL
LIN {X 0,Y 531,Z 355.336,A -85,B 0,C 180,E1 -4474.942,E2 -4474.942} C_VEL
LIN {X 0,Y 530.963,Z 355.34,A -85,B 0,C 180,E1 -4478.246,E2 -4478.246} C_VEL
LIN {X 0,Y 530.988,Z 355.338,A -85,B 0,C 180,E1 -4480.677,E2 -4480.677} C_VEL
LIN {X 0,Y 530.985,Z 355.338,A -85,B 0,C 180,E1 -4483.071,E2 -4483.071} C_VEL
LIN {X 0,Y 531.031,Z 355.341,A -85,B 0,C 180,E1 -4485.436,E2 -4485.436} C_VEL
LIN {X 0,Y 531.037,Z 355.33,A -85,B 0,C 180,E1 -4488.55,E2 -4488.55} C_VEL
LIN {X 0,Y 531.051,Z 355.333,A -85,B 0,C 180,E1 -4491.63,E2 -4491.63} C_VEL
LIN {X 0,Y 531.117,Z 355.322,A -85,B 0,C 180,E1 -4494.685,E2 -4494.685} C_VEL
LIN {X 0,Y 531.131,Z 355.322,A -85,B 0,C 180,E1 -4497.725,E2 -4497.725} C_VEL
LIN {X 0,Y 531.148,Z 355.32,A -85,B 0,C 180,E1 -4500.758,E2 -4500.758} C_VEL
LIN {X 0,Y 531.103,Z 355.326,A -85,B 0,C 180,E1 -4503.034,E2 -4503.034} C_VEL
LIN {X 0,Y 531.077,Z 355.326,A -85,B 0,C 180,E1 -4506.077,E2 -4506.077} C_VEL
LIN {X 0,Y 531.03,Z 355.34,A -85,B 0,C 180,E1 -4509.138,E2 -4509.138} C_VEL
LIN {X 0,Y 531.033,Z 355.33,A -85,B 0,C 180,E1 -4512.225,E2 -4512.225} C_VEL
LIN {X 0,Y 530.988,Z 355.342,A -85,B 0,C 180,E1 -4515.35,E2 -4515.35} C_VEL
LIN {X 0,Y 531.009,Z 355.337,A -85,B 0,C 180,E1 -4517.723,E2 -4517.723} C_VEL
LIN {X 0,Y 530.998,Z 355.342,A -85,B 0,C 180,E1 -4520.938,E2 -4520.938} C_VEL
LIN {X 0,Y 531.001,Z 355.334,A -85,B 0,C 180,E1 -4524.046,E2 -4524.046} C_VEL
LIN {X 0,Y 531.006,Z 355.342,A -85,B 0,C 180,E1 -4526.744,E2 -4526.744} C_VEL
LIN {X 0,Y 530.977,Z 355.343,A -85,B 0,C 180,E1 -4529.323,E2 -4529.323} C_VEL
LIN {X 0,Y 530.975,Z 355.341,A -85,B 0,C 180,E1 -4532.104,E2 -4532.104} C_VEL
LIN {X 0,Y 530.986,Z 355.342,A -85,B 0,C 180,E1 -4534.855,E2 -4534.855} C_VEL
LIN {X 0,Y 530.963,Z 355.342,A -85,B 0,C 180,E1 -4537.508,E2 -4537.508} C_VEL
LIN {X 0,Y 530.998,Z 355.341,A -85,B 0,C 180,E1 -4540.432,E2 -4540.432} C_VEL
LIN {X 0,Y 530.965,Z 355.342,A -85,B 0,C 180,E1 -4543.495,E2 -4543.495} C_VEL
LIN {X 0,Y 530.962,Z 355.343,A -85,B 0,C 180,E1 -4543.58,E2 -4543.58} C_VEL
LIN {X 0,Y 530.289,Z 355.429,A -85,B 0,C 180,E1 -4544.214,E2 -4544.214} C_VEL
LIN {X 0,Y 527.442,Z 355.788,A -85,B 0,C 180,E1 -4545.243,E2 -4545.243} C_VEL
LIN {X 0,Y 525.039,Z 356.09,A -85,B 0,C 180,E1 -4546.071,E2 -4546.071} C_VEL
LIN {X 0,Y 524.006,Z 356.216,A -85,B 0,C 180,E1 -4546.711,E2 -4546.711} C_VEL
LIN {X 0,Y 523.921,Z 356.223,A -85,B 0,C 180,E1 -4546.927,E2 -4546.927} C_VEL
LIN {X 0,Y 523.947,Z 356.217,A -85,B 0,C 180,E1 -4549.922,E2 -4549.922} C_VEL
LIN {X 0,Y 523.912,Z 356.229,A -85,B 0,C 180,E1 -4552.869,E2 -4552.869} C_VEL
LIN {X 0,Y 523.969,Z 356.323,A -85,B 0,C 180,E1 -4554.851,E2 -4554.851} C_VEL
LIN {X 0,Y 524.577,Z 360.565,A -85,B 0,C 180,E1 -4555.759,E2 -4555.759} C_VEL
LIN {X 0,Y 524.254,Z 376.107,A -85,B 0,C 180,E1 -4558.915,E2 -4558.915} C_VEL
LIN {X 0,Y 525.992,Z 385.741,A -85,B 0,C 180,E1 -4559.101,E2 -4559.101} C_VEL
LIN {X 0,Y 525.538,Z 482.477,A -85,B 0,C 180,E1 -4560.45,E2 -4560.45} C_VEL
LIN {X 0,Y 525.304,Z 495.855,A -85,B 0,C 180,E1 -4560.797,E2 -4560.797} C_VEL
LIN {X 0,Y 525.115,Z 508.857,A -85,B 0,C 180,E1 -4561.306,E2 -4561.306} C_VEL
LIN {X 0,Y 524.85,Z 520.765,A -85,B 0,C 180,E1 -4561.944,E2 -4561.944} C_VEL
LIN {X 0,Y 524.578,Z 531.614,A -85,B 0,C 180,E1 -4562.687,E2 -4562.687} C_VEL
LIN {X 0,Y 524.301,Z 541.578,A -85,B 0,C 180,E1 -4563.533,E2 -4563.533} C_VEL
LIN {X 0,Y 524.09,Z 549.969,A -85,B 0,C 180,E1 -4564.401,E2 -4564.401} C_VEL
LIN {X 0,Y 523.882,Z 558.164,A -85,B 0,C 180,E1 -4565.426,E2 -4565.426} C_VEL
LIN {X 0,Y 523.662,Z 566.188,A -85,B 0,C 180,E1 -4566.677,E2 -4566.677} C_VEL
LIN {X 0,Y 523.517,Z 572.515,A -85,B 0,C 180,E1 -4567.921,E2 -4567.921} C_VEL
LIN {X 0,Y 523.432,Z 577.405,A -85,B 0,C 180,E1 -4569.157,E2 -4569.157} C_VEL
LIN {X 0,Y 523.351,Z 581.031,A -85,B 0,C 180,E1 -4570.384,E2 -4570.384} C_VEL
LIN {X 0,Y 523.287,Z 582.797,A -85,B 0,C 180,E1 -4571.196,E2 -4571.196} C_VEL
LIN {X 0,Y 523.294,Z 584.671,A -85,B 0,C 180,E1 -4572.47,E2 -4572.47} C_VEL
LIN {X 0,Y 523.24,Z 585.435,A -85,B 0,C 180,E1 -4573.617,E2 -4573.617} C_VEL
LIN {X 0,Y 523.227,Z 585.447,A -85,B 0,C 180,E1 -4574.417,E2 -4574.417} C_VEL
LIN {X 0,Y 523.308,Z 585.041,A -85,B 0,C 180,E1 -4575.232,E2 -4575.232} C_VEL
LIN {X 0,Y 523.307,Z 584.217,A -85,B 0,C 180,E1 -4576.011,E2 -4576.011} C_VEL
LIN {X 0,Y 523.294,Z 582.956,A -85,B 0,C 180,E1 -4576.802,E2 -4576.802} C_VEL
LIN {X 0,Y 523.395,Z 580.261,A -85,B 0,C 180,E1 -4577.988,E2 -4577.988} C_VEL
LIN {X 0,Y 523.434,Z 576.546,A -85,B 0,C 180,E1 -4579.166,E2 -4579.166} C_VEL
LIN {X 0,Y 523.522,Z 571.706,A -85,B 0,C 180,E1 -4580.34,E2 -4580.34} C_VEL
LIN {X 0,Y 523.654,Z 565.61,A -85,B 0,C 180,E1 -4581.51,E2 -4581.51} C_VEL
LIN {X 0,Y 523.881,Z 557.755,A -85,B 0,C 180,E1 -4582.717,E2 -4582.717} C_VEL
LIN {X 0,Y 524.104,Z 548.555,A -85,B 0,C 180,E1 -4583.842,E2 -4583.842} C_VEL
LIN {X 0,Y 524.338,Z 538.799,A -85,B 0,C 180,E1 -4584.809,E2 -4584.809} C_VEL
LIN {X 0,Y 524.65,Z 527.86,A -85,B 0,C 180,E1 -4585.679,E2 -4585.679} C_VEL
LIN {X 0,Y 524.921,Z 517.172,A -85,B 0,C 180,E1 -4586.354,E2 -4586.354} C_VEL
LIN {X 0,Y 525.22,Z 504.3,A -85,B 0,C 180,E1 -4586.98,E2 -4586.98} C_VEL
LIN {X 0,Y 525.403,Z 491.928,A -85,B 0,C 180,E1 -4587.413,E2 -4587.413} C_VEL
LIN {X 0,Y 525.548,Z 479.036,A -85,B 0,C 180,E1 -4587.701,E2 -4587.701} C_VEL
LIN {X 0,Y 525.89,Z 384.578,A -85,B 0,C 180,E1 -4589.007,E2 -4589.007} C_VEL
LIN {X 0,Y 524.163,Z 375.814,A -85,B 0,C 180,E1 -4589.184,E2 -4589.184} C_VEL
LIN {X 0,Y 524.511,Z 362.45,A -85,B 0,C 180,E1 -4591.92,E2 -4591.92} C_VEL
LIN {X 0,Y 524.472,Z 358.743,A -85,B 0,C 180,E1 -4592.688,E2 -4592.688} C_VEL
LIN {X 0,Y 524.011,Z 356.216,A -85,B 0,C 180,E1 -4593.268,E2 -4593.268} C_VEL
LIN {X 0,Y 524.033,Z 356.207,A -85,B 0,C 180,E1 -4596.159,E2 -4596.159} C_VEL
LIN {X 0,Y 523.999,Z 356.217,A -85,B 0,C 180,E1 -4599.262,E2 -4599.262} C_VEL
LIN {X 0,Y 524.009,Z 356.211,A -85,B 0,C 180,E1 -4601.739,E2 -4601.739} C_VEL
LIN {X 0,Y 523.999,Z 356.213,A -85,B 0,C 180,E1 -4605.052,E2 -4605.052} C_VEL
LIN {X 0,Y 523.968,Z 356.213,A -85,B 0,C 180,E1 -4607.968,E2 -4607.968} C_VEL
LIN {X 0,Y 523.976,Z 356.211,A -85,B 0,C 180,E1 -4610.409,E2 -4610.409} C_VEL
LIN {X 0,Y 523.921,Z 356.221,A -85,B 0,C 180,E1 -4612.893,E2 -4612.893} C_VEL
LIN {X 0,Y 523.957,Z 356.22,A -85,B 0,C 180,E1 -4615.418,E2 -4615.418} C_VEL
LIN {X 0,Y 523.97,Z 356.212,A -85,B 0,C 180,E1 -4617.998,E2 -4617.998} C_VEL
LIN {X 0,Y 523.949,Z 356.219,A -85,B 0,C 180,E1 -4620.854,E2 -4620.854} C_VEL
LIN {X 0,Y 523.963,Z 356.214,A -85,B 0,C 180,E1 -4623.734,E2 -4623.734} C_VEL
LIN {X 0,Y 523.924,Z 356.218,A -85,B 0,C 180,E1 -4626.403,E2 -4626.403} C_VEL
LIN {X 0,Y 523.924,Z 356.227,A -85,B 0,C 180,E1 -4629.083,E2 -4629.083} C_VEL
LIN {X 0,Y 523.955,Z 356.213,A -85,B 0,C 180,E1 -4632.117,E2 -4632.117} C_VEL
LIN {X 0,Y 523.954,Z 356.219,A -85,B 0,C 180,E1 -4635.308,E2 -4635.308} C_VEL
LIN {X 0,Y 523.959,Z 356.218,A -85,B 0,C 180,E1 -4638.688,E2 -4638.688} C_VEL
LIN {X 0,Y 523.913,Z 356.219,A -85,B 0,C 180,E1 -4641.897,E2 -4641.897} C_VEL
LIN {X 0,Y 523.934,Z 356.226,A -85,B 0,C 180,E1 -4644.908,E2 -4644.908} C_VEL
LIN {X 0,Y 523.938,Z 356.216,A -85,B 0,C 180,E1 -4647.677,E2 -4647.677} C_VEL
LIN {X 0,Y 523.949,Z 356.221,A -85,B 0,C 180,E1 -4650.675,E2 -4650.675} C_VEL
LIN {X 0,Y 523.971,Z 356.212,A -85,B 0,C 180,E1 -4653.728,E2 -4653.728} C_VEL
LIN {X 0,Y 523.929,Z 356.219,A -85,B 0,C 180,E1 -4656.27,E2 -4656.27} C_VEL
LIN {X 0,Y 523.94,Z 356.225,A -85,B 0,C 180,E1 -4658.766,E2 -4658.766} C_VEL
LIN {X 0,Y 523.947,Z 356.217,A -85,B 0,C 180,E1 -4661.22,E2 -4661.22} C_VEL
LIN {X 0,Y 523.933,Z 356.216,A -85,B 0,C 180,E1 -4663.638,E2 -4663.638} C_VEL
LIN {X 0,Y 523.932,Z 356.217,A -85,B 0,C 180,E1 -4666.028,E2 -4666.028} C_VEL
LIN {X 0,Y 524.003,Z 356.213,A -85,B 0,C 180,E1 -4668.394,E2 -4668.394} C_VEL
LIN {X 0,Y 523.999,Z 356.208,A -85,B 0,C 180,E1 -4671.516,E2 -4671.516} C_VEL
LIN {X 0,Y 524.09,Z 356.206,A -85,B 0,C 180,E1 -4674.614,E2 -4674.614} C_VEL
LIN {X 0,Y 524.103,Z 356.195,A -85,B 0,C 180,E1 -4677.694,E2 -4677.694} C_VEL
LIN {X 0,Y 524.116,Z 356.199,A -85,B 0,C 180,E1 -4680.768,E2 -4680.768} C_VEL
LIN {X 0,Y 524.067,Z 356.201,A -85,B 0,C 180,E1 -4683.075,E2 -4683.075} C_VEL
LIN {X 0,Y 524.037,Z 356.208,A -85,B 0,C 180,E1 -4686.159,E2 -4686.159} C_VEL
LIN {X 0,Y 523.994,Z 356.209,A -85,B 0,C 180,E1 -4689.262,E2 -4689.262} C_VEL
LIN {X 0,Y 523.998,Z 356.209,A -85,B 0,C 180,E1 -4691.743,E2 -4691.743} C_VEL
LIN {X 0,Y 523.983,Z 356.211,A -85,B 0,C 180,E1 -4695.053,E2 -4695.053} C_VEL
LIN {X 0,Y 523.955,Z 356.217,A -85,B 0,C 180,E1 -4697.969,E2 -4697.969} C_VEL
LIN {X 0,Y 523.964,Z 356.22,A -85,B 0,C 180,E1 -4700.41,E2 -4700.41} C_VEL
LIN {X 0,Y 523.909,Z 356.221,A -85,B 0,C 180,E1 -4702.894,E2 -4702.894} C_VEL
LIN {X 0,Y 523.946,Z 356.215,A -85,B 0,C 180,E1 -4705.419,E2 -4705.419} C_VEL
LIN {X 0,Y 523.963,Z 356.219,A -85,B 0,C 180,E1 -4707.999,E2 -4707.999} C_VEL
LIN {X 0,Y 523.945,Z 356.216,A -85,B 0,C 180,E1 -4710.857,E2 -4710.857} C_VEL
LIN {X 0,Y 523.956,Z 356.217,A -85,B 0,C 180,E1 -4713.736,E2 -4713.736} C_VEL
LIN {X 0,Y 523.916,Z 356.223,A -85,B 0,C 180,E1 -4716.405,E2 -4716.405} C_VEL
LIN {X 0,Y 523.954,Z 356.214,A -85,B 0,C 180,E1 -4719.082,E2 -4719.082} C_VEL
LIN {X 0,Y 523.953,Z 356.222,A -85,B 0,C 180,E1 -4722.119,E2 -4722.119} C_VEL
LIN {X 0,Y 523.952,Z 356.215,A -85,B 0,C 180,E1 -4725.309,E2 -4725.309} C_VEL
LIN {X 0,Y 523.969,Z 356.213,A -85,B 0,C 180,E1 -4728.688,E2 -4728.688} C_VEL
LIN {X 0,Y 523.951,Z 356.214,A -85,B 0,C 180,E1 -4731.076,E2 -4731.076} C_VEL
LIN {X 0,Y 523.927,Z 356.225,A -85,B 0,C 180,E1 -4733.828,E2 -4733.828} C_VEL
LIN {X 0,Y 523.942,Z 356.216,A -85,B 0,C 180,E1 -4736.637,E2 -4736.637} C_VEL
LIN {X 0,Y 523.964,Z 356.215,A -85,B 0,C 180,E1 -4739.357,E2 -4739.357} C_VEL
LIN {X 0,Y 523.98,Z 356.218,A -85,B 0,C 180,E1 -4742.281,E2 -4742.281} C_VEL
LIN {X 0,Y 524.029,Z 356.235,A -85,B 0,C 180,E1 -4744.905,E2 -4744.905} C_VEL
LIN {X 0,Y 525.635,Z 365.057,A -85,B 0,C 180,E1 -4746.353,E2 -4746.353} C_VEL
LIN {X 0,Y 525.168,Z 382.546,A -85,B 0,C 180,E1 -4749.025,E2 -4749.025} C_VEL
LIN {X 0,Y 524.686,Z 402.745,A -85,B 0,C 180,E1 -4752.057,E2 -4752.057} C_VEL
LIN {X 0,Y 524.335,Z 421.505,A -85,B 0,C 180,E1 -4754.839,E2 -4754.839} C_VEL
LIN {X 0,Y 525.962,Z 432.953,A -85,B 0,C 180,E1 -4755.047,E2 -4755.047} C_VEL
LIN {X 0,Y 525.521,Z 529.955,A -85,B 0,C 180,E1 -4756.392,E2 -4756.392} C_VEL
LIN {X 0,Y 525.275,Z 543.287,A -85,B 0,C 180,E1 -4756.73,E2 -4756.73} C_VEL
LIN {X 0,Y 525.018,Z 556.62,A -85,B 0,C 180,E1 -4757.24,E2 -4757.24} C_VEL
LIN {X 0,Y 524.714,Z 568.976,A -85,B 0,C 180,E1 -4757.894,E2 -4757.894} C_VEL
LIN {X 0,Y 524.474,Z 580.746,A -85,B 0,C 180,E1 -4758.699,E2 -4758.699} C_VEL
LIN {X 0,Y 524.166,Z 590.974,A -85,B 0,C 180,E1 -4759.572,E2 -4759.572} C_VEL
LIN {X 0,Y 523.953,Z 600.181,A -85,B 0,C 180,E1 -4760.543,E2 -4760.543} C_VEL
LIN {X 0,Y 523.732,Z 609.154,A -85,B 0,C 180,E1 -4761.706,E2 -4761.706} C_VEL
LIN {X 0,Y 523.583,Z 616.377,A -85,B 0,C 180,E1 -4762.868,E2 -4762.868} C_VEL
LIN {X 0,Y 523.508,Z 622.959,A -85,B 0,C 180,E1 -4764.221,E2 -4764.221} C_VEL
LIN {X 0,Y 523.36,Z 627.309,A -85,B 0,C 180,E1 -4765.379,E2 -4765.379} C_VEL
LIN {X 0,Y 523.443,Z 629.618,A -85,B 0,C 180,E1 -4766.151,E2 -4766.151} C_VEL
LIN {X 0,Y 523.367,Z 631.484,A -85,B 0,C 180,E1 -4766.921,E2 -4766.921} C_VEL
LIN {X 0,Y 523.334,Z 632.884,A -85,B 0,C 180,E1 -4767.691,E2 -4767.691} C_VEL
LIN {X 0,Y 523.25,Z 634.49,A -85,B 0,C 180,E1 -4769.23,E2 -4769.23} C_VEL
LIN {X 0,Y 523.249,Z 634.707,A -85,B 0,C 180,E1 -4770,E2 -4770} C_VEL
LIN {X 0,Y 523.274,Z 633.881,A -85,B 0,C 180,E1 -4771.539,E2 -4771.539} C_VEL
LIN {X 0,Y 523.334,Z 632.885,A -85,B 0,C 180,E1 -4772.309,E2 -4772.309} C_VEL
LIN {X 0,Y 523.367,Z 631.484,A -85,B 0,C 180,E1 -4773.079,E2 -4773.079} C_VEL
LIN {X 0,Y 523.424,Z 628.538,A -85,B 0,C 180,E1 -4774.235,E2 -4774.235} C_VEL
LIN {X 0,Y 523.461,Z 624.548,A -85,B 0,C 180,E1 -4775.393,E2 -4775.393} C_VEL
LIN {X 0,Y 523.517,Z 619.298,A -85,B 0,C 180,E1 -4776.576,E2 -4776.576} C_VEL
LIN {X 0,Y 523.651,Z 612.95,A -85,B 0,C 180,E1 -4777.713,E2 -4777.713} C_VEL
LIN {X 0,Y 523.835,Z 604.891,A -85,B 0,C 180,E1 -4778.875,E2 -4778.875} C_VEL
LIN {X 0,Y 524.034,Z 596.68,A -85,B 0,C 180,E1 -4779.845,E2 -4779.845} C_VEL
LIN {X 0,Y 524.344,Z 586.672,A -85,B 0,C 180,E1 -4780.815,E2 -4780.815} C_VEL
LIN {X 0,Y 524.56,Z 575.402,A -85,B 0,C 180,E1 -4781.689,E2 -4781.689} C_VEL
LIN {X 0,Y 524.861,Z 564.304,A -85,B 0,C 180,E1 -4782.371,E2 -4782.371} C_VEL
LIN {X 0,Y 525.107,Z 552.042,A -85,B 0,C 180,E1 -4782.954,E2 -4782.954} C_VEL
LIN {X 0,Y 525.349,Z 539.169,A -85,B 0,C 180,E1 -4783.391,E2 -4783.391} C_VEL
LIN {X 0,Y 525.563,Z 525.515,A -85,B 0,C 180,E1 -4783.681,E2 -4783.681} C_VEL
LIN {X 0,Y 525.804,Z 431.229,A -85,B 0,C 180,E1 -4784.98,E2 -4784.98} C_VEL
LIN {X 0,Y 524.313,Z 421.401,A -85,B 0,C 180,E1 -4785.166,E2 -4785.166} C_VEL
LIN {X 0,Y 524.711,Z 401.43,A -85,B 0,C 180,E1 -4788.123,E2 -4788.123} C_VEL
LIN {X 0,Y 525.147,Z 382.42,A -85,B 0,C 180,E1 -4790.976,E2 -4790.976} C_VEL
LIN {X 0,Y 525.575,Z 364.896,A -85,B 0,C 180,E1 -4793.65,E2 -4793.65} C_VEL
LIN {X 0,Y 524.029,Z 356.21,A -85,B 0,C 180,E1 -4795.095,E2 -4795.095} C_VEL
LIN {X 0,Y 523.97,Z 356.22,A -85,B 0,C 180,E1 -4797.998,E2 -4797.998} C_VEL
LIN {X 0,Y 523.952,Z 356.216,A -85,B 0,C 180,E1 -4800.856,E2 -4800.856} C_VEL
LIN {X 0,Y 523.96,Z 356.217,A -85,B 0,C 180,E1 -4803.734,E2 -4803.734} C_VEL
LIN {X 0,Y 523.921,Z 356.224,A -85,B 0,C 180,E1 -4806.404,E2 -4806.404} C_VEL
LIN {X 0,Y 523.957,Z 356.213,A -85,B 0,C 180,E1 -4809.08,E2 -4809.08} C_VEL
LIN {X 0,Y 523.969,Z 356.214,A -85,B 0,C 180,E1 -4811.312,E2 -4811.312} C_VEL
LIN {X 0,Y 523.952,Z 356.215,A -85,B 0,C 180,E1 -4814.691,E2 -4814.691} C_VEL
LIN {X 0,Y 523.953,Z 356.222,A -85,B 0,C 180,E1 -4817.881,E2 -4817.881} C_VEL
LIN {X 0,Y 523.954,Z 356.214,A -85,B 0,C 180,E1 -4820.918,E2 -4820.918} C_VEL
LIN {X 0,Y 523.922,Z 356.226,A -85,B 0,C 180,E1 -4823.827,E2 -4823.827} C_VEL
LIN {X 0,Y 523.937,Z 356.215,A -85,B 0,C 180,E1 -4826.635,E2 -4826.635} C_VEL
LIN {X 0,Y 523.956,Z 356.217,A -85,B 0,C 180,E1 -4829.356,E2 -4829.356} C_VEL
LIN {X 0,Y 523.972,Z 356.213,A -85,B 0,C 180,E1 -4832.28,E2 -4832.28} C_VEL
LIN {X 0,Y 523.946,Z 356.214,A -85,B 0,C 180,E1 -4834.581,E2 -4834.581} C_VEL
LIN {X 0,Y 523.908,Z 356.222,A -85,B 0,C 180,E1 -4837.106,E2 -4837.106} C_VEL
LIN {X 0,Y 523.97,Z 356.218,A -85,B 0,C 180,E1 -4839.865,E2 -4839.865} C_VEL
LIN {X 0,Y 523.962,Z 356.211,A -85,B 0,C 180,E1 -4842.837,E2 -4842.837} C_VEL
LIN {X 0,Y 523.995,Z 356.214,A -85,B 0,C 180,E1 -4845.236,E2 -4845.236} C_VEL
LIN {X 0,Y 524.002,Z 356.207,A -85,B 0,C 180,E1 -4848.394,E2 -4848.394} C_VEL
